REGION Network 7: INITIALIZE ALL STATIONS TIMER
   #tmrInitAllStns(IN := "HMI".settings.kp8.buttons[0].actuate, PT := t#10s);   // TON
   #initAllStns := #tmrInitAllStns.Q;
END_REGION

REGION Network 8: SET DEFAULT TIMERS
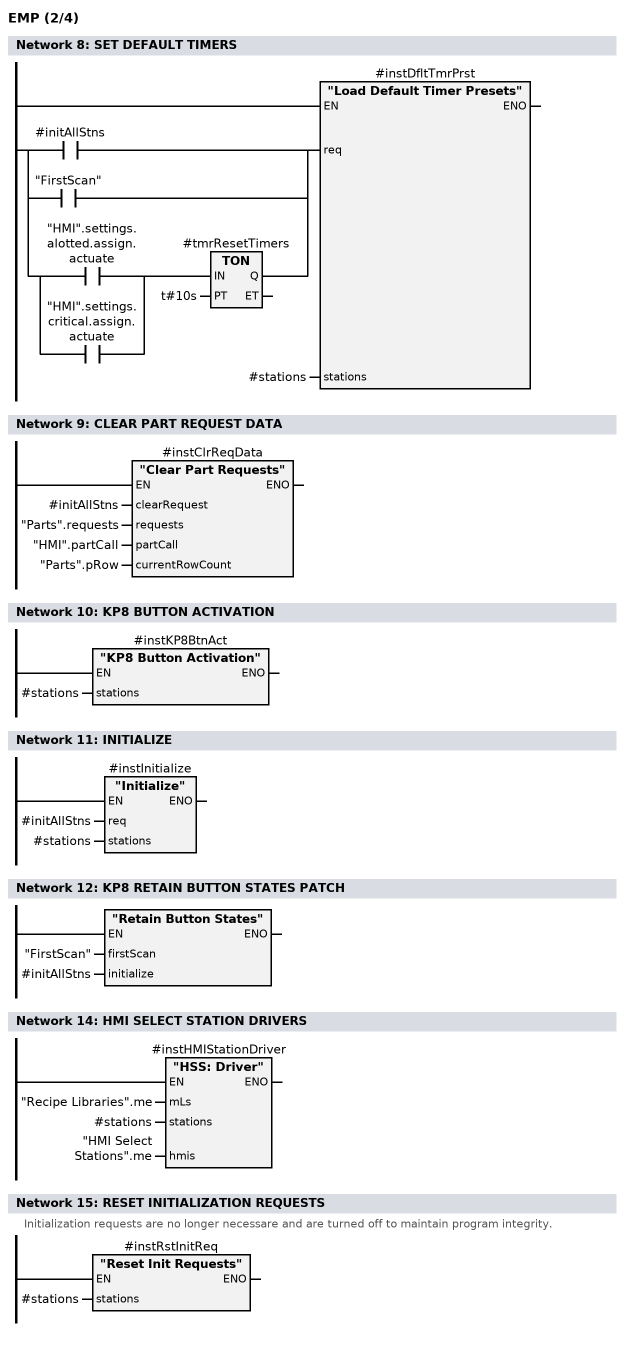
   #tmrResetTimers(IN := "HMI".settings.alotted.assign.actuate OR "HMI".settings.critical.assign.actuate,   // TON
                   PT := t#10s);
   #instDfltTmrPrst(req := #initAllStns OR "FirstScan" OR #tmrResetTimers.Q, stations := #stations);   // "Load Default Timer Presets"
END_REGION

REGION Network 9: CLEAR PART REQUEST DATA
   RUNG wire#powerrail
      #instClrReqData(clearRequest := #initAllStns, requests := "Parts".requests, partCall := "HMI".partCall, currentRowCount := "Parts".pRow)
   END_RUNG
   // the same network as SCL:
   #instClrReqData(clearRequest := #initAllStns,   // "Clear Part Requests"
                   requests := "Parts".requests,
                   partCall := "HMI".partCall,
                   currentRowCount := "Parts".pRow);
END_REGION

REGION Network 10: KP8 BUTTON ACTIVATION
   RUNG wire#powerrail
      #instKP8BtnAct(stations := #stations)
   END_RUNG
   // the same network as SCL:
   #instKP8BtnAct(stations := #stations);   // "KP8 Button Activation"
END_REGION

REGION Network 11: INITIALIZE
   RUNG wire#powerrail
      #instInitialize(req := #initAllStns, stations := #stations)
   END_RUNG
   // the same network as SCL:
   #instInitialize(req := #initAllStns, stations := #stations);   // "Initialize"
END_REGION

REGION Network 12: KP8 RETAIN BUTTON STATES PATCH
   RUNG wire#powerrail
      "Retain Button States"(firstScan := "FirstScan", initialize := #initAllStns)
   END_RUNG
   // the same network as SCL:
   "Retain Button States"(firstScan := "FirstScan", initialize := #initAllStns);
END_REGION

REGION Network 13 (SCL): KP8 DRIVER CALLS
   REGION "LOOP THROUGH STATIONS"
       FOR #i := 0 TO "stnCount" DO
           CASE #i OF
               0..24, 30..38:
                   #instKP8Drvs[#i](btnIn := #stations.me[#i].kp8In,
                                    hardInit := #stations.me[#i].init.hard,
                                    softInit := #stations.me[#i].init.soft,
                                    btn0Activate := #stations.me[#i].kp8Config.activate[0],
                                    btn0Mode := #stations.me[#i].kp8Config.mode[0],
                                    btn0Group := #stations.me[#i].kp8Config.group[0],
                                    btn0Flash := #stations.me[#i].kp8Config.flash[0],
                                    btn0ColorOn1 := #stations.me[#i].kp8Config.colorOn1[0],
                                    btn0ColorOn2 := #stations.me[#i].kp8Config.colorOn2[0],
                                    btn0ColorOff := #stations.me[#i].kp8Config.colorOff[0],
                                    btn1Activate := #stations.me[#i].kp8Config.activate[1],
                                    btn1Mode := #stations.me[#i].kp8Config.mode[1],
                                    btn1Group := #stations.me[#i].kp8Config.group[1],
                                    btn1Flash := #stations.me[#i].kp8Config.flash[1],
                                    btn1ColorOn1 := #stations.me[#i].kp8Config.colorOn1[1],
                                    btn1ColorOn2 := #stations.me[#i].kp8Config.colorOn2[1],
                                    btn1ColorOff := #stations.me[#i].kp8Config.colorOff[1],
                                    btn2Activate := #stations.me[#i].kp8Config.activate[2],
                                    btn2Mode := #stations.me[#i].kp8Config.mode[2],
                                    btn2Group := #stations.me[#i].kp8Config.group[2],
                                    btn2Flash := #stations.me[#i].kp8Config.flash[2],
                                    btn2ColorOn1 := #stations.me[#i].kp8Config.colorOn1[2],
                                    btn2ColorOn2 := #stations.me[#i].kp8Config.colorOn2[2],
                                    btn2ColorOff := #stations.me[#i].kp8Config.colorOff[2],
                                    btn3Activate := #stations.me[#i].kp8Config.activate[3],
                                    btn3Mode := #stations.me[#i].kp8Config.mode[3],
                                    btn3Group := #stations.me[#i].kp8Config.group[3],
                                    btn3Flash := #stations.me[#i].kp8Config.flash[3],
                                    btn3ColorOn1 := #stations.me[#i].kp8Config.colorOn1[3],
                                    btn3ColorOn2 := #stations.me[#i].kp8Config.colorOn2[3],
                                    btn3ColorOff := #stations.me[#i].kp8Config.colorOff[3],
                                    btn4Activate := #stations.me[#i].kp8Config.activate[4],
                                    btn4Mode := #stations.me[#i].kp8Config.mode[4],
                                    btn4Group := #stations.me[#i].kp8Config.group[4],
                                    btn4Flash := #stations.me[#i].kp8Config.flash[4],
                                    btn4ColorOn1 := #stations.me[#i].kp8Config.colorOn1[4],
                                    btn4ColorOn2 := #stations.me[#i].kp8Config.colorOn2[4],
                                    btn4ColorOff := #stations.me[#i].kp8Config.colorOff[4],
                                    btn5Activate := #stations.me[#i].kp8Config.activate[5],
                                    btn5Mode := #stations.me[#i].kp8Config.mode[5],
                                    btn5Group := #stations.me[#i].kp8Config.group[5],
                                    btn5Flash := #stations.me[#i].kp8Config.flash[5],
                                    btn5ColorOn1 := #stations.me[#i].kp8Config.colorOn1[5],
                                    btn5ColorOn2 := #stations.me[#i].kp8Config.colorOn2[5],
                                    btn5ColorOff := #stations.me[#i].kp8Config.colorOff[5],
                                    btn6Activate := #stations.me[#i].kp8Config.activate[6],
                                    btn6Mode := #stations.me[#i].kp8Config.mode[6],
                                    btn6Group := #stations.me[#i].kp8Config.group[6],
                                    btn6Flash := #stations.me[#i].kp8Config.flash[6],
                                    btn6ColorOn1 := #stations.me[#i].kp8Config.colorOn1[6],
                                    btn6ColorOn2 := #stations.me[#i].kp8Config.colorOn2[6],
                                    btn6ColorOff := #stations.me[#i].kp8Config.colorOff[6],
                                    btn7Activate := #stations.me[#i].kp8Config.activate[7],
                                    btn7Mode := #stations.me[#i].kp8Config.mode[7],
                                    btn7Group := #stations.me[#i].kp8Config.group[7],
                                    btn7Flash := #stations.me[#i].kp8Config.flash[7],
                                    btn7ColorOn1 := #stations.me[#i].kp8Config.colorOn1[7],
                                    btn7ColorOn2 := #stations.me[#i].kp8Config.colorOn2[7],
                                    btn7ColorOff := #stations.me[#i].kp8Config.colorOff[7],
                                    btnStatesOut => #stations.me[#i].btnStates,
                                    btnColorsOut => #stations.me[#i].kp8Out);
               ELSE 
                   ;
           END_CASE;

       END_FOR;
   END_REGION
END_REGION

REGION Network 14: HMI SELECT STATION DRIVERS
   RUNG wire#powerrail
      #instHMIStationDriver(mLs := "Recipe Libraries".me, stations := #stations, hmis := "HMI Select Stations".me)
   END_RUNG
   // the same network as SCL:
   #instHMIStationDriver(mLs := "Recipe Libraries".me, stations := #stations, hmis := "HMI Select Stations".me);   // "HSS: Driver"
END_REGION

REGION Network 15: RESET INITIALIZATION REQUESTS
   // Initialization requests are no longer necessare and are turned off to maintain program integrity.
   RUNG wire#powerrail
      #instRstInitReq(stations := #stations)
   END_RUNG
   // the same network as SCL:
   #instRstInitReq(stations := #stations);   // "Reset Init Requests"
END_REGION

REGION Network 16: BARCODE SCREEN
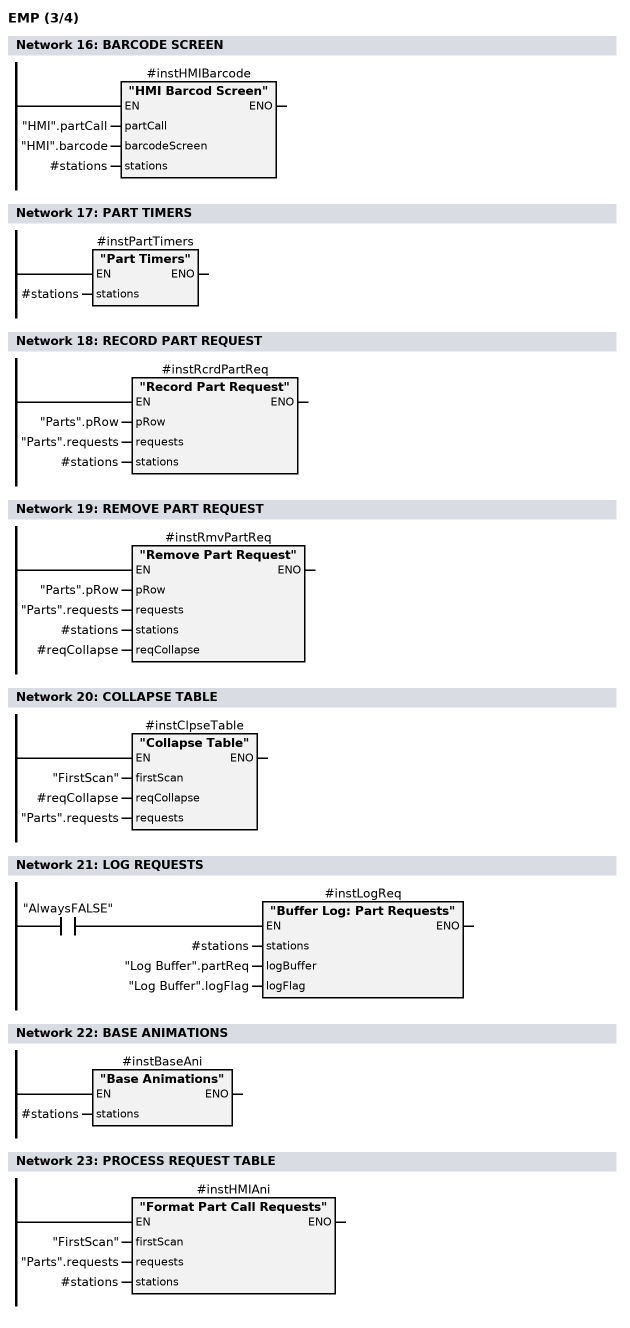
   RUNG wire#powerrail
      #instHMIBarcode(partCall := "HMI".partCall, barcodeScreen := "HMI".barcode, stations := #stations)
   END_RUNG
   // the same network as SCL:
   #instHMIBarcode(partCall := "HMI".partCall, barcodeScreen := "HMI".barcode, stations := #stations);   // "HMI Barcod Screen"
END_REGION

REGION Network 17: PART TIMERS
   RUNG wire#powerrail
      #instPartTimers(stations := #stations)
   END_RUNG
   // the same network as SCL:
   #instPartTimers(stations := #stations);   // "Part Timers"
END_REGION

REGION Network 18: RECORD PART REQUEST
   RUNG wire#powerrail
      #instRcrdPartReq(pRow := "Parts".pRow, requests := "Parts".requests, stations := #stations)
   END_RUNG
   // the same network as SCL:
   #instRcrdPartReq(pRow := "Parts".pRow, requests := "Parts".requests, stations := #stations);   // "Record Part Request"
END_REGION

REGION Network 19: REMOVE PART REQUEST
   RUNG wire#powerrail
      #instRmvPartReq(pRow := "Parts".pRow, requests := "Parts".requests, stations := #stations, reqCollapse := #reqCollapse)
   END_RUNG
   // the same network as SCL:
   #instRmvPartReq(pRow := "Parts".pRow,   // "Remove Part Request"
                   requests := "Parts".requests,
                   stations := #stations,
                   reqCollapse := #reqCollapse);
END_REGION

REGION Network 20: COLLAPSE TABLE
   RUNG wire#powerrail
      #instClpseTable(firstScan := "FirstScan", reqCollapse := #reqCollapse, requests := "Parts".requests)
   END_RUNG
   // the same network as SCL:
   #instClpseTable(firstScan := "FirstScan", reqCollapse := #reqCollapse, requests := "Parts".requests);   // "Collapse Table"
END_REGION

REGION Network 21: LOG REQUESTS
   RUNG wire#powerrail
      Contact( "AlwaysFALSE" )
      #instLogReq(stations := #stations, logBuffer := "Log Buffer".partReq, logFlag := "Log Buffer".logFlag)
   END_RUNG
   // the same network as SCL:
   IF "AlwaysFALSE" THEN
       #instLogReq(stations := #stations, logBuffer := "Log Buffer".partReq, logFlag := "Log Buffer".logFlag);   // "Buffer Log: Part Requests"
   END_IF;
END_REGION

REGION Network 22: BASE ANIMATIONS
   RUNG wire#powerrail
      #instBaseAni(stations := #stations)
   END_RUNG
   // the same network as SCL:
   #instBaseAni(stations := #stations);   // "Base Animations"
END_REGION

REGION Network 23: PROCESS REQUEST TABLE
   RUNG wire#powerrail
      #instHMIAni(firstScan := "FirstScan", requests := "Parts".requests, stations := #stations)
   END_RUNG
   // the same network as SCL:
   #instHMIAni(firstScan := "FirstScan", requests := "Parts".requests, stations := #stations);   // "Format Part Call Requests"
END_REGION

REGION Network 24: HMI POPULATE TABLE
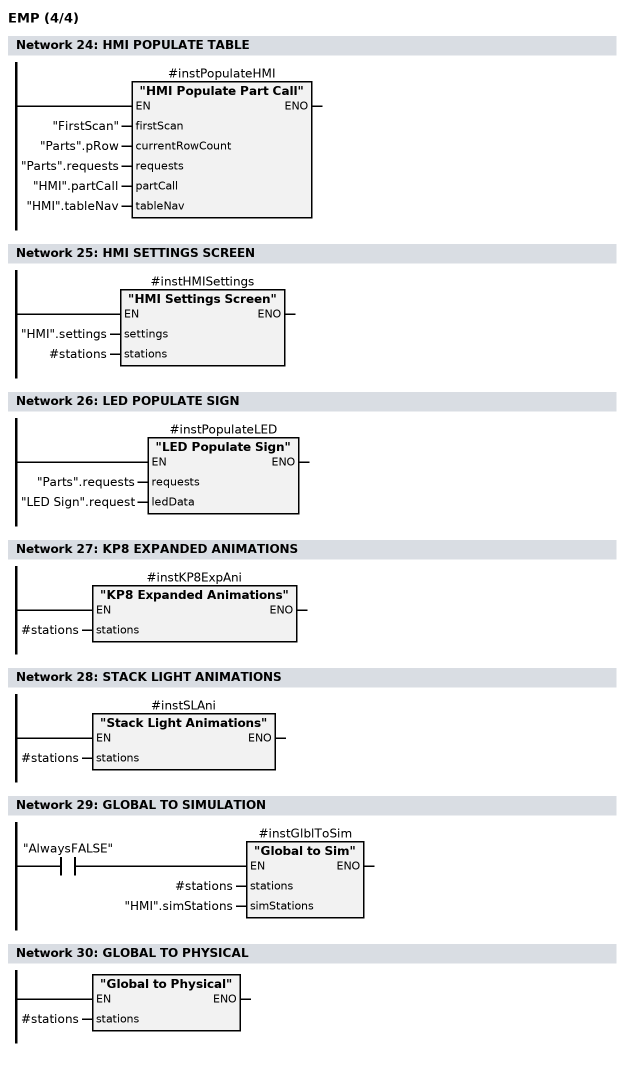
   RUNG wire#powerrail
      #instPopulateHMI(firstScan := "FirstScan", currentRowCount := "Parts".pRow, requests := "Parts".requests, partCall := "HMI".partCall, tableNav := "HMI".tableNav)
   END_RUNG
   // the same network as SCL:
   #instPopulateHMI(firstScan := "FirstScan",   // "HMI Populate Part Call"
                    currentRowCount := "Parts".pRow,
                    requests := "Parts".requests,
                    partCall := "HMI".partCall,
                    tableNav := "HMI".tableNav);
END_REGION

REGION Network 25: HMI SETTINGS SCREEN
   RUNG wire#powerrail
      #instHMISettings(settings := "HMI".settings, stations := #stations)
   END_RUNG
   // the same network as SCL:
   #instHMISettings(settings := "HMI".settings, stations := #stations);   // "HMI Settings Screen"
END_REGION

REGION Network 26: LED POPULATE SIGN
   RUNG wire#powerrail
      #instPopulateLED(requests := "Parts".requests, ledData := "LED Sign".request)
   END_RUNG
   // the same network as SCL:
   #instPopulateLED(requests := "Parts".requests, ledData := "LED Sign".request);   // "LED Populate Sign"
END_REGION

REGION Network 27: KP8 EXPANDED ANIMATIONS
   RUNG wire#powerrail
      #instKP8ExpAni(stations := #stations)
   END_RUNG
   // the same network as SCL:
   #instKP8ExpAni(stations := #stations);   // "KP8 Expanded Animations"
END_REGION

REGION Network 28: STACK LIGHT ANIMATIONS
   RUNG wire#powerrail
      #instSLAni(stations := #stations)
   END_RUNG
   // the same network as SCL:
   #instSLAni(stations := #stations);   // "Stack Light Animations"
END_REGION

REGION Network 29: GLOBAL TO SIMULATION
   RUNG wire#powerrail
      Contact( "AlwaysFALSE" )
      #instGlblToSim(stations := #stations, simStations := "HMI".simStations)
   END_RUNG
   // the same network as SCL:
   IF "AlwaysFALSE" THEN
       #instGlblToSim(stations := #stations, simStations := "HMI".simStations);   // "Global to Sim"
   END_IF;
END_REGION

REGION Network 30: GLOBAL TO PHYSICAL
   RUNG wire#powerrail
      "Global to Physical"(stations := #stations)
   END_RUNG
   // the same network as SCL:
   "Global to Physical"(stations := #stations);
END_REGION
END_FUNCTION_BLOCK

FUNCTION_BLOCK "Code 128"   // FB2, SCL
{ S7_Optimized_Access := 'TRUE' }
VERSION : 0.1
   VAR_INPUT
      partNumber : String;
   END_VAR
   VAR_OUTPUT
      barcode : String;
   END_VAR
   VAR
      charsIn : Array[0..255] of Byte;
      charsOut : Array[0..255] of Byte;
      cnt : UInt;
      intVals : Array[0..255] of Int;
      sum : Int;
      checkSum : Int;
   END_VAR
   VAR_TEMP
      pn : String;
      i : Int;
   END_VAR
   VAR CONSTANT
      startChar : Char := 'Ì';
      stopChar : Char := 'Î';
   END_VAR
   // intVals[0] := 104;
BEGIN
   #pn := #partNumber;

   FOR #i := 0 TO 255 DO
       #charsIn[#i] := 16#00;
       #charsOut[#i] := 16#00;
       #intVals[#i] := 0;
   END_FOR;

   Strg_TO_Chars(Strg:=#pn,
                 pChars:=0,
                 Cnt=>#cnt,
                 Chars:=#charsIn);


   #sum := 104;
   FOR #i := 0 TO UINT_TO_INT(#cnt - 1) DO
       #intVals[#i] := CHAR_TO_INT(#charsIn[#i]) - 32;
       #intVals[#i] := #intVals[#i] * (#i + 1);
       #sum := #sum + #intVals[#i];
   END_FOR;
   #checkSum := (#sum MOD 103) + 32;
   IF #checkSum >= 127 THEN
       #checkSum := #checkSum + 68;
   END_IF;

   #charsOut[0] := #startChar;
   FOR #i := 1 TO UINT_TO_INT(#cnt) DO
       #charsOut[#i] := #charsIn[#i - 1];
   END_FOR;
   #charsOut[#cnt + 1] := INT_TO_BYTE(#checkSum);
   #charsOut[#cnt + 2] := INT_TO_BYTE(#stopChar);

   Chars_TO_Strg(Chars := #charsOut,
                 pChars := 0,
                 Cnt := #cnt + 3,
                 Strg => #barcode);
END_FUNCTION_BLOCK

FUNCTION_BLOCK "HMI Barcod Screen"   // FB3, SCL
{ S7_Optimized_Access := 'TRUE' }
VERSION : 0.1
   VAR_IN_OUT
      partCall : "Part Call Screen";
      barcodeScreen : "Barcode Screen";
      stations : "Stations";
   END_VAR
   VAR
      address : UInt;
      button : UInt;
      instCode128 : "Code 128";
      codeOut : String;
      pnOut : WString[40];
      station : UInt;
      oldSelectedRow : Int;
      oldOrderedBtn : Bool;
   END_VAR
   VAR_TEMP
      orderCancelled : Int;
      processedPN : String[40];
      selectedPN : String[40];
      userOrdered : Bool;
      selectedRow : Int;
      position : Int;
   END_VAR
   VAR CONSTANT
      maxRows : Int := 199;
   END_VAR
BEGIN
   REGION "GET USER ROW SELECTION"
       #selectedRow := "Get Part Call Row Number"(partCall := #partCall); 
   END_REGION

   REGION "ON SELECTION OF A PART CALL ROW
       IF #selectedRow <> 0 THEN
           IF #selectedRow <> #oldSelectedRow THEN

               REGION "GET BUTTON AND STATION NUMBERS"
                   #address := #partCall.row[#selectedRow - 1].address;
                   "Address to Station and Button"(address := #address,
                                                   station => #station,
                                                   button => #button);
               END_REGION

               REGION "CONVERT STRING TO BARCODE"

                   REGION "COPY TO LOCALS"
                       #selectedPN := WSTRING_TO_STRING(#partCall.row[#selectedRow - 1].tfPartNumber.value);
                   END_REGION

                   REGION "CHECK FOR MULTI LINE"

                       REGION "GET POSITON OF CARRIAGE RETURN"
                           #position := FIND(IN1 := #selectedPN, IN2 := '$L');
                       END_REGION

                       REGION "MULTILINE"
                           IF #position <> 0 THEN
                               #processedPN := LEFT(IN := #selectedPN, L := #position - 1);
                           END_IF;
                       END_REGION

                       REGION "SINGLE LINE"
                           IF #position = 0 THEN
                               #processedPN := #selectedPN;
                           END_IF;
                       END_REGION

                   END_REGION

                   REGION "CONVERT TO BARCODE"
                       #instCode128(partNumber := #processedPN,
                                    barcode => #codeOut);
                   END_REGION

                   REGION "OUTPUT FOR HMI SCREEN"
                       #barcodeScreen.partNumber := STRING_TO_WSTRING(#processedPN);
                       #barcodeScreen.barcode := #codeOut;
                   END_REGION

               END_REGION

           END_IF;
       END_IF;
   END_REGION

   REGION "PASS USER ORDERED"

       REGION "COPY TO LOCAL"
           #userOrdered := #barcodeScreen.ordered;
       END_REGION

       REGION "TURN OFF THE LIGHTS"
           #barcodeScreen.ordered := FALSE;
       END_REGION

       REGION "ON RISING EDGE"
           IF #userOrdered AND NOT #oldOrderedBtn THEN

               REGION "SET PART ORDERED"
                   #stations.me[#station - 1].partOrdered[#button - 1] := #userOrdered;
               END_REGION

           END_IF;
       END_REGION

       REGION "CHANGE DETECTION"
           #oldOrderedBtn := #userOrdered;
       END_REGION

   END_REGION

   REGION "CHANGE DETECTION"    
       #oldSelectedRow := #selectedRow;
   END_REGION
END_FUNCTION_BLOCK

FUNCTION_BLOCK "Initialize"   // FB4, SCL
{ S7_Optimized_Access := 'TRUE' }
VERSION : 0.1
   VAR_INPUT
      req : Bool;
   END_VAR
   VAR_IN_OUT
      stations : "Stations";
   END_VAR
   VAR
      rtElapsed : Real;
      rt : "Runtime Data";
   END_VAR
   VAR_TEMP
      i : Int;
      reset : Struct
         req : Bool;
         elapsed : Real;
      END_STRUCT;
      init : Bool;
   END_VAR
   VAR CONSTANT
      resetLimit : Real := 1.25;
   END_VAR
BEGIN
   REGION "FIRST SCAN OR REQUEST"
       IF #req THEN
           // initialize all stations on plc first scan
           FOR #i := 0 TO "stnCount" DO
               #stations.me[#i].init.hard := TRUE;
           END_FOR;
       END_IF;
   END_REGION

   REGION "RUNTIME CALL"
       // get elapsed time
       #rt.elapsed := RUNTIME(#rt.mem);
       // convert to real data type
       #rtElapsed := LREAL_TO_REAL(#rt.elapsed);
   END_REGION

   REGION "BUTTON 0 BASED RESET TIMERS"
       FOR #i := 0 TO "stnCount" DO

           REGION "PRE-CONDITION"
               // init off by default
               #init := FALSE;
               // request is button 0 on kp8
               #reset.req := #stations.me[#i].kp8In.%X0;
               // saved to shorter name
               #reset.elapsed := #stations.me[#i].elapsedTime.resetReq;
           END_REGION

           REGION "RESET REQUEST"
               IF NOT #reset.req THEN
                   #reset.elapsed := 0.0;
               END_IF;
               IF #reset.req THEN
                   // incriment elapsed time
                   #reset.elapsed := #reset.elapsed + #rtElapsed;
                   // timer expired condition
                   IF #reset.elapsed >= #resetLimit THEN
                       #init := TRUE;
                       #reset.elapsed := 0.0;
                   END_IF;
               END_IF;
               // save elapsed time
               #stations.me[#i].elapsedTime.resetReq := #reset.elapsed;
           END_REGION

           REGION "SAVE INITIALIZATIN REQUEST"
               #stations.me[#i].init.hard := #init;
           END_REGION

       END_FOR;
   END_REGION
END_FUNCTION_BLOCK

FUNCTION_BLOCK "Reset Init Requests"   // FB5, SCL
{ S7_Optimized_Access := 'TRUE' }
VERSION : 0.1
   VAR_IN_OUT
      stations : "Stations";
   END_VAR
   VAR
      placeHolder : Bool;
   END_VAR
   VAR_TEMP
      i : Int;
      stnCount : Int;
   END_VAR
BEGIN
   REGION "GET STATION COUNT"
       #stnCount := "stnCount";
   END_REGION

   REGION "RESET INITIALIZATION REQUESTS
       FOR #i := 0 TO #stnCount DO
           #stations.me[#i].init.hard := FALSE;
           #stations.me[#i].init.soft := FALSE;
       END_FOR;
   END_REGION
END_FUNCTION_BLOCK

FUNCTION_BLOCK "Record Part Request"   // FB6, SCL
{ S7_Optimized_Access := 'TRUE' }
VERSION : 0.1
   VAR_IN_OUT
      pRow : Int;
      requests : "Part Request Data";
      stations : "Stations";
   END_VAR
   VAR
      enterAddress : Bool;
      old : Struct
         presses : "Station Old Presses";
      END_STRUCT;
   END_VAR
   VAR_TEMP
      address : UInt;
      hasPart : Bool;
      i : Int;
      j : Int;
      k : Int;
      logAddress : UInt;
      noPart : Bool;
      oldPartReq : Bool;
      partReq : Bool;
      partNumber : WString;
   END_VAR
BEGIN
   REGION "FOR EACH STATION"
       FOR #i := 0 TO "stnCount" DO

           REGION "FOR EACH BUTTON"
               // j = 0 is excluded because it is used as a station reset button
               FOR #j := 1 TO "ptsPerStn" DO

                   REGION "COPY TO LOCAL"
                       #partReq := #stations.me[#i].btnStates[#j];
                       #oldPartReq := #old.presses.me[#i,#j];
                   END_REGION

                   REGION "DETERMINE STATE"

                       REGION "ON NEW REQUEST"
                           IF #partReq AND NOT #oldPartReq THEN

                               REGION "COPY TO LOCAL"
                                   #partNumber := #stations.me[#i].partNumbers[#j];
                               END_REGION

                               REGION "BUTTON HAS NO PN"
                                   IF LEN(#partNumber) = 0 THEN
                                       #hasPart := FALSE;
                                       #noPart := TRUE;
                                   END_IF;
                               END_REGION

                               REGION "BUTTON HAS PN"
                                   IF LEN(#partNumber) <> 0 THEN
                                       #hasPart := TRUE;
                                       #noPart := FALSE;
                                   END_IF;
                               END_REGION

                           END_IF;

                           REGION "SAVE FOR CHANGE DETECTION"
                               #old.presses.me[#i, #j] := #stations.me[#i].btnStates[#j];
                           END_REGION

                       END_REGION

                   END_REGION

                   REGION "NO PART"
                       IF #noPart THEN

                           REGION "TURN OFF THE LIGHTS"
                               #hasPart := FALSE;
                               #noPart := FALSE;
                               #enterAddress := FALSE;
                           END_REGION

                       END_IF;
                   END_REGION

                   REGION "HAS PART"
                       IF #hasPart THEN

                           REGION "TURN OFF THE LIGHTS"
                               #hasPart := FALSE;
                               #noPart := FALSE;
                               #enterAddress := FALSE;
                           END_REGION

                           REGION "CALCULATE ADDRESS"
                               #address := (INT_TO_UINT(#i) + 1) * 10 + (INT_TO_UINT(#j) + 1);
                           END_REGION

                           REGION "SET FLAG"
                               #enterAddress := TRUE;
                           END_REGION

                           REGION "CHECK FOR ENTRY IN DB"
                               REGION "FOR EACH ROW IN PART DB"
                                   FOR #k := 0 TO "partReqDataRowCount" DO

                                       REGION "COPY TO LOCAL"
                                           #logAddress := #requests.row[#k].address;
                                       END_REGION

                                       REGION "RESET FLAG"
                                           IF #logAddress = #address THEN
                                               #enterAddress := FALSE;
                                           END_IF;
                                       END_REGION

                                   END_FOR;
                               END_REGION
                           END_REGION


                       END_IF;
                   END_REGION

                   REGION "SAVE ROW DATA"
                       IF #enterAddress THEN

                           REGION "TURN OFF THE LIGHTS"
                               #enterAddress := FALSE;
                           END_REGION

                           REGION "ENTER PART REQUEST"
                               #stations.me[#i].partRequested[#j] := TRUE;
                           END_REGION

                           REGION "ADDRESS"
                               #requests.row[#pRow].address := #address;
                           END_REGION

                           REGION "LINE"
                               #requests.row[#pRow].tfLine.value := #stations.me[#i].line;
                           END_REGION

                           REGION "DROP ZONE"
                               #requests.row[#pRow].tfDropZone.value := USINT_TO_WSTRING(#stations.me[#i].dropZone);
                           END_REGION

                           REGION "PART NUMBER"
                               #requests.row[#pRow].tfPartNumber.value := #stations.me[#i].partNumbers[#j];
                           END_REGION

                           REGION "ELLAPSED TIME"
                               #requests.row[#pRow].tfTime.value := "Real to WString Timer"(#stations.me[#i].elapsedTime.partReq[#j]);
                           END_REGION

                           REGION "ROW POINTER"

                               REGION "INCREMENT"
                                   #pRow := #pRow + 1;
                               END_REGION

                               REGION "HIGH LIMIT ROLLOVER"
                                   IF #pRow > "partReqDataRowCount" THEN
                                       #pRow := 0;
                                   END_IF;
                               END_REGION

                           END_REGION

                       END_IF;
                   END_REGION

               END_FOR;
           END_REGION

       END_FOR;
   END_REGION
END_FUNCTION_BLOCK

FUNCTION_BLOCK "Part Timers"   // FB7, SCL
{ S7_Optimized_Access := 'TRUE' }
VERSION : 0.1
   VAR_IN_OUT
      stations : "Stations";
   END_VAR
   VAR
      rt : "Runtime Data";
      old : Struct
         presses : "Station Old Presses";
      END_STRUCT;
   END_VAR
   VAR_TEMP
      alottedTime : Real;
      btnCount : Int;
      elapsedTime : Real;
      i : Int;
      j : Int;
      partRequested : Bool;
      redTime : Real;
      remainingTime : Real;
      stnCount : Int;
      press : Struct
         current : Bool;
         old : Bool;
      END_STRUCT;
   END_VAR
BEGIN
   REGION "RUNTIME CALL"
       #rt.elapsed := RUNTIME(#rt.mem);
       #rt.asReal := LREAL_TO_REAL(#rt.elapsed);
   END_REGION

   REGION "COPY TO LOCAL"
       #stnCount := "stnCount";
       #btnCount := "ptsPerStn";
   END_REGION

   REGION "FOR EACH STATION"
       FOR #i := 0 TO #stnCount DO

           REGION "FOR EACH BUTTON"
               // j := 0 would be the reset button so it is skipped
               FOR #j := 1 TO #btnCount DO

                   REGION "RESET PART TIMER"

                       REGION "COPY TO LOCAL"
                           #press.current := #stations.me[#i].btnStates[#j];
                           #press.old := #old.presses.me[#i, #j];
                       END_REGION

                       REGION "ON PRESS FALLING EDGE"
                           IF NOT #press.current AND #press.old THEN
                               #stations.me[#i].elapsedTime.partReq[#j] := 0.0;
                           END_IF;
                           #old.presses.me[#i, #j] := #stations.me[#i].btnStates[#j];
                       END_REGION

                   END_REGION

                   REGION "PART REQUEST TIMER"

                       REGION "COPY TO LOCAL"
                           #partRequested := #stations.me[#i].btnStates[#j];
                       END_REGION

                       REGION "ON PART REQUEST"
                           IF #partRequested THEN

                               REGION "OUTPUT ELLAPSED TIME"
                                   // get saved time
                                   #elapsedTime := #stations.me[#i].elapsedTime.partReq[#j];
                                   // add elapsed time
                                   #elapsedTime += #rt.asReal;
                                   // save new value
                                   #stations.me[#i].elapsedTime.partReq[#j] := #elapsedTime;
                               END_REGION

                           END_IF;
                       END_REGION

                   END_REGION

               END_FOR;
           END_REGION

       END_FOR;
   END_REGION
END_FUNCTION_BLOCK

FUNCTION_BLOCK "Base Animations"   // FB8, SCL
{ S7_Optimized_Access := 'TRUE' }
VERSION : 0.1
   VAR_IN_OUT
      stations : "Stations";
   END_VAR
   VAR_TEMP
      animation : Int;
      i : Int;
      j : Int;
      partRequested : Bool;
      partOrdered : Bool;
      elapsedTime : Real;
      criticalTime : Real;
      alottedTime : Real;
      remainingTime : Real;
      stnCount : Int;
   END_VAR
   VAR CONSTANT
      anDefault : USInt := 0;
      anRequested : USInt := 1;
      anSolidRed : USInt := 2;
      anFlashRed : USInt := 3;
      anPartOrdered : USInt := 4;
   END_VAR
BEGIN
   REGION "COPY TO LOCAL"
       #stnCount := "stnCount";
   END_REGION

   REGION "FOR EACH STATION"
       FOR #i := 0 TO #stnCount DO

           REGION "FOR EACH BUTTON"
               // j := 0 would be the reset button so it is skipped
               FOR #j := 1 TO 7 DO

                   REGION "PART REQUEST TIMER"

                       REGION "COPY TO LOCAL"
                           #partRequested := #stations.me[#i].btnStates[#j];
                           #partOrdered := #stations.me[#i].partOrdered[#j];
                       END_REGION

                       REGION "PART REQUESTED"
                           IF #partRequested THEN

                               REGION "COPY TO LOCAL"
                                   // remaining time
                                   #elapsedTime := #stations.me[#i].elapsedTime.partReq[#j];
                                   #alottedTime := #stations.me[#i].presetTime.allotted[#j];
                                   #remainingTime := #alottedTime - #elapsedTime;
                                   // critical time
                                   #criticalTime := #stations.me[#i].presetTime.critical[#j];
                               END_REGION

                               REGION "DEFAULT ANIMATION STATE"
                                   IF #remainingTime > #criticalTime THEN
                                       #animation := #anRequested;
                                   END_IF;
                               END_REGION

                               REGION "ORDERED"
                                   IF #partOrdered THEN
                                       #animation := #anPartOrdered;
                                   END_IF;
                               END_REGION

                               REGION "SOLID RED ANIMATION STATE"
                                   IF #remainingTime <= #criticalTime AND #elapsedTime > 0.0 THEN
                                       #animation := #anSolidRed;
                                   END_IF;
                               END_REGION

                               REGION "FLASHING RED ANIMATION STATE
                                   IF #remainingTime <= 0.0 THEN
                                       #animation := #anFlashRed;
                                   END_IF;
                               END_REGION

                           END_IF;
                       END_REGION

                       REGION "PART NOT REQUESTED"
                           IF NOT #partRequested THEN
                               #animation := #anDefault;
                           END_IF;
                       END_REGION

                       REGION "OUTPUT"
                           #stations.me[#i].animations[#j] := #animation;
                       END_REGION

                   END_REGION

               END_FOR;
           END_REGION

       END_FOR;
   END_REGION
END_FUNCTION_BLOCK

FUNCTION_BLOCK "Format Part Call Requests"   // FB9, SCL
{ S7_Optimized_Access := 'TRUE' }
VERSION : 0.1
   VAR_INPUT
      firstScan : Bool;
   END_VAR
   VAR_IN_OUT
      requests : "Part Request Data";
      stations : "Stations";
   END_VAR
   VAR
      station : Int;
      button : Int;
   END_VAR
   VAR_TEMP
      address : Int;
      animate : USInt;
      timeAsReal : Real;
      timeAsTime : WString;
      i : Int;
      inStrRslt : Int;
      invisible : USInt;
      genericVisible : USInt;
      gray : USInt;
      darkGray : USInt;
      red : USInt;
      blue : USInt;
      redFlashing : USInt;
   END_VAR
   VAR CONSTANT
      visible : USInt := 1;
      anDefault : USInt := 0;
      anRequested : USInt := 1;
      anSolidRed : USInt := 2;
      anFlashRed : USInt := 3;
      anPartOrdered : USInt := 4;
   END_VAR
BEGIN
   REGION "COPY TO LOCAL"
       #invisible := "invisible";
       #gray := "BgGray";
       #darkGray := "disabled";
       #blue := "BgLBl";
       #red := "BgDRd";
       #redFlashing := "FlDrd";
   END_REGION


   REGION "ITERATE THROUGH VISIBLE TABLE ROWS"
       FOR #i := 0 TO "partReqDataRowCount" DO

           REGION "COPY TO LOCAL"
               #address := UINT_TO_INT(#requests.row[#i].address);
           END_REGION

           REGION "HIDE UNPOPULATED ROWS"
               IF #address = 0 THEN
                   #requests.row[#i].pbSelection.animate := #invisible;
                   #requests.row[#i].rtBackground.animate := #invisible;
                   #animate := 0;
                   #requests.row[#i].tfDropZone.animate := #invisible;
                   #requests.row[#i].tfLine.animate := #invisible;
                   #requests.row[#i].tfPartNumber.animateSL := #invisible;
                   #requests.row[#i].tfPartNumber.animateDL := #invisible;
                   #requests.row[#i].tfTime.animate := #invisible;
               END_IF;
           END_REGION

           REGION "ANIMATE POPULATED ROWS"

               REGION "ANIMATE ROWS WITH DATA"
                   IF #address <> 0 THEN

                       REGION "GET POINTERS FOR STATION ARRAY"
                           #station := #address / 10 - 1;
                           #button := #address MOD 10 - 1;
                       END_REGION

                       REGION "SET ANIMATE"
                           CASE #stations.me[#station].animations[#button] OF
                               #anRequested:
                                   #animate := #gray;
                               #anSolidRed:
                                   #animate := #red;
                               #anFlashRed:
                                   #animate := #redFlashing;
                               #anPartOrdered:
                                   #animate := #blue;
                               ELSE
                                   #animate := #invisible;
                           END_CASE;
                       END_REGION


                       REGION "ANIMATIONS"

                           REGION "PUSHBUTTON VISIBILITY"
                               #requests.row[#i].pbSelection.animate := #visible;
                           END_REGION

                           REGION "BACKGROUND VISIBILITY"
                               #requests.row[#i].rtBackground.animate := #darkGray;
                           END_REGION

                           REGION "DROP ZONE" 
                               #requests.row[#i].tfDropZone.animate := #animate;
                               #requests.row[#i].tfDropZone.value := "Strip Sign"(UINT_TO_WSTRING(#stations.me[#station].dropZone));
                           END_REGION

                           REGION "LINE"
                               #requests.row[#i].tfLine.animate := #animate;
                               #requests.row[#i].tfLine.value := #stations.me[#station].line;
                           END_REGION

                           REGION "PART NUMBER"
                               #requests.row[#i].tfPartNumber.animateSL := #animate;
                               #requests.row[#i].tfPartNumber.value := #stations.me[#station].partNumbers[#button];
                               REGION "DETERMINE VISIBLE ROWS"

                                   REGION "FIND CARRIAGE RETURN"
                                       #inStrRslt := FIND(IN1 := #requests.row[#i].tfPartNumber.value,
                                                          IN2 := wstring#'$L');
                                   END_REGION

                                   REGION "SINGLE LINE"
                                       IF #inStrRslt = 0 THEN
                                           #requests.row[#i].tfPartNumber.animateSL := #animate;
                                           #requests.row[#i].tfPartNumber.animateDL := #invisible;
                                       END_IF;
                                   END_REGION

                                   REGION "DOUBLE LINE"
                                       IF #inStrRslt <> 0 THEN
                                           #requests.row[#i].tfPartNumber.animateSL := #invisible;
                                           #requests.row[#i].tfPartNumber.animateDL := #animate;
                                       END_IF;
                                   END_REGION

                               END_REGION

                           END_REGION

                           REGION "TIME"
                               #requests.row[#i].tfTime.animate := #animate;
                               #timeAsReal := #stations.me[#station].presetTime.allotted[#button];
                               #timeAsReal -= #stations.me[#station].elapsedTime.partReq[#button];
                               #requests.row[#i].tfTime.value := "Real to WString Timer"(#timeAsReal);
                           END_REGION

                       END_REGION

                   END_IF;
               END_REGION

           END_REGION

       END_FOR;
   END_REGION
END_FUNCTION_BLOCK

FUNCTION_BLOCK "KP8 Expanded Animations"   // FB10, SCL
{ S7_Optimized_Access := 'TRUE' }
VERSION : 0.1
   VAR_IN_OUT
      stations : "Stations";
   END_VAR
   VAR_TEMP
      i : Int;
      j : Int;
      colorBox : DWord;
      animation : Int;
      mask : DWord;
   END_VAR
   VAR CONSTANT
      anSolidRed : USInt := 2;
      anFlashRed : USInt := 3;
      anBlue : USInt := 4;
   END_VAR
BEGIN
   REGION "LOOP THROUGH STATIONS"
       FOR #i := 0 TO "stnCount" DO

           REGION "LOOP THROUGH BUTTONS"
               FOR #j := 0 TO "ptsPerStn" DO

                   REGION "GET ANIMATION"
                       #animation := #stations.me[#i].animations[#j];
                   END_REGION

                   REGION "SOLID RED"
                       IF #animation = #anSolidRed THEN
                           #colorBox := #stations.me[#i].kp8Out;
                           #mask := 16#FEFEFEFF;
                           #mask := ROL_DWORD(IN := #mask,
                                                 N := INT_TO_UINT(#j));
                           #colorBox := #colorBox AND #mask;
                           #mask := 16#100_0000;
                           #mask := ROL_DWORD(IN := #mask,
                                                 N := INT_TO_UINT(#j));
                           #colorBox := #colorBox OR #mask;
                           #stations.me[#i].kp8Out := #colorBox;
                       END_IF;
                   END_REGION

                   REGION "FLASHING RED"
                       IF #animation = #anFlashRed THEN

                           REGION "RED ON"
                               IF "Clock_1Hz" THEN
                                   #colorBox := #stations.me[#i].kp8Out;
                                   #mask := 16#FEFEFEFF;
                                   #mask := ROL_DWORD(IN := #mask,
                                                         N := INT_TO_UINT(#j));
                                   #colorBox := #colorBox AND #mask;
                                   #mask := 16#100_0000;
                                   #mask := ROL_DWORD(IN := #mask,
                                                         N := INT_TO_UINT(#j));
                                   #colorBox := #colorBox OR #mask;
                                   #stations.me[#i].kp8Out := #colorBox;
                               END_IF;
                           END_REGION

                           REGION "RED OFF"
                               IF NOT "Clock_1Hz" THEN
                                   #colorBox := #stations.me[#i].kp8Out;
                                   #mask := 16#FEFEFEFF;
                                   #mask := ROL_DWORD(IN := #mask,
                                                         N := INT_TO_UINT(#j));
                                   #colorBox := #colorBox AND #mask;
                                   #stations.me[#i].kp8Out := #colorBox;
                               END_IF;
                           END_REGION

                       END_IF;
                   END_REGION

                   REGION "BLUE"
                       IF #animation = #anBlue THEN
                           #colorBox := #stations.me[#i].kp8Out;
                           #mask := 16#FEFEFEFF;
                           #mask := ROL_DWORD(IN := #mask,
                                              N := INT_TO_UINT(#j));
                           #colorBox := #colorBox AND #mask;
                           #mask := 16#0000_0100;
                           #mask := ROL_DWORD(IN := #mask,
                                                 N := INT_TO_UINT(#j));
                           #colorBox := #colorBox OR #mask;
                           #stations.me[#i].kp8Out := #colorBox;
                       END_IF;
                   END_REGION

               END_FOR;
           END_REGION

       END_FOR;
   END_REGION
END_FUNCTION_BLOCK

FUNCTION_BLOCK "Stack Light Animations"   // FB11, SCL
{ S7_Optimized_Access := 'TRUE' }
VERSION : 0.1
   VAR_IN_OUT
      stations : "Stations";
   END_VAR
   VAR_TEMP
      animation : Int;
      i : Int;
      j : Int;
      stackLight : DWord;
   END_VAR
   VAR CONSTANT
      anDefault : USInt := 0;
      anRequested : USInt := 1;
      anSolidRed : USInt := 2;
      anFlashRed : USInt := 3;
      anPartOrdered : USInt := 4;
      buttonCount : Int := 7;
      "Part 01" : Int := 7;
      "Part 01 Green On" : DWord := 16#0400_0000;
      "Part 01 Red On" : DWord := 16#0100_0000;
      "Part 01 Yellow On" : DWord := 16#0200_0000;
      "Part 02" : Int := 3;
      "Part 02 Green On" : DWord := 16#2000_0000;
      "Part 02 Red On" : DWord := 16#0800_0000;
      "Part 02 Yellow On" : DWord := 16#1000_0000;
      "Part 03" : Int := 6;
      "Part 03 Green On" : DWord := 16#0001_0000;
      "Part 03 Red On" : DWord := 16#4000_0000;
      "Part 03 Yellow On" : DWord := 16#8000_0000;
      "Part 04" : Int := 2;
      "Part 04 Green On" : DWord := 16#0008_0000;
      "Part 04 Yellow On" : DWord := 16#0004_0000;
      "Part 04 Red On" : DWord := 16#0002_0000;
      "Part 05" : Int := 5;
      "Part 05 Green On" : DWord := 16#0040_0000;
      "Part 05 Red On" : DWord := 16#0010_0000;
      "Part 05 Yellow On" : DWord := 16#0020_0000;
      "Part 06" : Int := 1;
      "Part 06 Green On" : DWord := 16#0000_0200;
      "Part 06 Red On" : DWord := 16#0080_0000;
      "Part 06 Yellow On" : DWord := 16#0000_0100;
   END_VAR
BEGIN
   REGION "LOOP THROUGH STATIONS"
       FOR #i := 0 TO "stnCount" DO

           REGION "LOOP THROUGH BUTTONS"
               FOR #j := 0 TO #buttonCount DO

                   REGION "COPY INTO LOCAL"
                       #stackLight := #stations.me[#i].stackLightOut;
                       #animation := #stations.me[#i].animations[#j];
                   END_REGION

                   REGION "GREEN"
                       IF #animation = #anDefault THEN
                           CASE #j OF
                               #"Part 01":
                                   #stackLight := #stackLight AND (NOT #"Part 01 Red On");
                                   #stackLight := #stackLight AND (NOT #"Part 01 Yellow On");
                                   #stackLight := #stackLight OR #"Part 01 Green On";
                               #"Part 02":
                                   #stackLight := #stackLight AND (NOT #"Part 02 Red On");
                                   #stackLight := #stackLight AND (NOT #"Part 02 Yellow On");
                                   #stackLight := #stackLight OR #"Part 02 Green On";
                               #"Part 03":
                                   #stackLight := #stackLight AND (NOT #"Part 03 Red On");
                                   #stackLight := #stackLight AND (NOT #"Part 03 Yellow On");
                                   #stackLight := #stackLight OR #"Part 03 Green On";
                               #"Part 04":
                                   #stackLight := #stackLight AND (NOT #"Part 04 Red On");
                                   #stackLight := #stackLight AND (NOT #"Part 04 Yellow On");
                                   #stackLight := #stackLight OR #"Part 04 Green On";
                               #"Part 05":
                                   #stackLight := #stackLight AND (NOT #"Part 05 Red On");
                                   #stackLight := #stackLight AND (NOT #"Part 05 Yellow On");
                                   #stackLight := #stackLight OR #"Part 05 Green On";
                               #"Part 06":
                                   #stackLight := #stackLight AND (NOT #"Part 06 Red On");
                                   #stackLight := #stackLight AND (NOT #"Part 06 Yellow On");
                                   #stackLight := #stackLight OR #"Part 06 Green On";
                               ELSE
                                   ;
                           END_CASE;
                       END_IF;
                   END_REGION

                   REGION "OFF"
                       IF #stations.me[#i].partNumbers[#j] = WSTRING#'' THEN
                           CASE #j OF
                               #"Part 01":
                                   #stackLight := #stackLight AND (NOT #"Part 01 Red On");
                                   #stackLight := #stackLight AND (NOT #"Part 01 Yellow On");
                                   #stackLight := #stackLight AND (NOT #"Part 01 Green On");
                               #"Part 02":
                                   #stackLight := #stackLight AND (NOT #"Part 02 Red On");
                                   #stackLight := #stackLight AND (NOT #"Part 02 Yellow On");
                                   #stackLight := #stackLight AND (NOT #"Part 02 Green On");
                               #"Part 03":
                                   #stackLight := #stackLight AND (NOT #"Part 03 Red On");
                                   #stackLight := #stackLight AND (NOT #"Part 03 Yellow On");
                                   #stackLight := #stackLight AND (NOT #"Part 03 Green On");
                               #"Part 04":
                                   #stackLight := #stackLight AND (NOT #"Part 04 Red On");
                                   #stackLight := #stackLight AND (NOT #"Part 04 Yellow On");
                                   #stackLight := #stackLight AND (NOT #"Part 04 Green On");
                               #"Part 05":
                                   #stackLight := #stackLight AND (NOT #"Part 05 Red On");
                                   #stackLight := #stackLight AND (NOT #"Part 05 Yellow On");
                                   #stackLight := #stackLight AND (NOT #"Part 05 Green On");
                               #"Part 06":
                                   #stackLight := #stackLight AND (NOT #"Part 06 Red On");
                                   #stackLight := #stackLight AND (NOT #"Part 06 Yellow On");
                                   #stackLight := #stackLight AND (NOT #"Part 06 Green On");
                               ELSE
                                   ;
                           END_CASE;
                       END_IF;
                   END_REGION

                   REGION "YELLOW"
                       IF #animation = #anRequested THEN
                           CASE #j OF
                               #"Part 01":
                                   #stackLight := #stackLight AND (NOT #"Part 01 Red On");
                                   #stackLight := #stackLight OR #"Part 01 Yellow On";
                                   #stackLight := #stackLight AND (NOT #"Part 01 Green On");
                               #"Part 02":
                                   #stackLight := #stackLight AND (NOT #"Part 02 Red On");
                                   #stackLight := #stackLight OR #"Part 02 Yellow On";
                                   #stackLight := #stackLight AND (NOT #"Part 02 Green On");
                               #"Part 03":
                                   #stackLight := #stackLight AND (NOT #"Part 03 Red On");
                                   #stackLight := #stackLight OR #"Part 03 Yellow On";
                                   #stackLight := #stackLight AND (NOT #"Part 03 Green On");
                               #"Part 04":
                                   #stackLight := #stackLight AND (NOT #"Part 04 Red On");
                                   #stackLight := #stackLight OR #"Part 04 Yellow On";
                                   #stackLight := #stackLight AND (NOT #"Part 04 Green On");
                               #"Part 05":
                                   #stackLight := #stackLight AND (NOT #"Part 05 Red On");
                                   #stackLight := #stackLight OR #"Part 05 Yellow On";
                                   #stackLight := #stackLight AND (NOT #"Part 05 Green On");
                               #"Part 06":
                                   #stackLight := #stackLight AND (NOT #"Part 06 Red On");
                                   #stackLight := #stackLight OR #"Part 06 Yellow On";
                                   #stackLight := #stackLight AND (NOT #"Part 06 Green On");
                               ELSE
                                   ;
                           END_CASE;
                       END_IF;
                   END_REGION

                   REGION "SOLID RED"
                       IF #animation = #anSolidRed THEN
                           CASE #j OF
                               #"Part 01":
                                   #stackLight := #stackLight OR #"Part 01 Red On";
                                   #stackLight := #stackLight AND (NOT #"Part 01 Yellow On");
                                   #stackLight := #stackLight AND (NOT #"Part 01 Green On");
                               #"Part 02":
                                   #stackLight := #stackLight OR #"Part 02 Red On";
                                   #stackLight := #stackLight AND (NOT #"Part 02 Yellow On");
                                   #stackLight := #stackLight AND (NOT #"Part 02 Green On");
                               #"Part 03":
                                   #stackLight := #stackLight OR #"Part 03 Red On";
                                   #stackLight := #stackLight AND (NOT #"Part 03 Yellow On");
                                   #stackLight := #stackLight AND (NOT #"Part 03 Green On");
                               #"Part 04":
                                   #stackLight := #stackLight OR #"Part 04 Red On";
                                   #stackLight := #stackLight AND (NOT #"Part 04 Yellow On");
                                   #stackLight := #stackLight AND (NOT #"Part 04 Green On");
                               #"Part 05":
                                   #stackLight := #stackLight OR #"Part 05 Red On";
                                   #stackLight := #stackLight AND (NOT #"Part 05 Yellow On");
                                   #stackLight := #stackLight AND (NOT #"Part 05 Green On");
                               #"Part 06":
                                   #stackLight := #stackLight OR #"Part 06 Red On";
                                   #stackLight := #stackLight AND (NOT #"Part 06 Yellow On");
                                   #stackLight := #stackLight AND (NOT #"Part 06 Green On");
                               ELSE
                                   ;
                           END_CASE;
                       END_IF;
                   END_REGION

                   REGION "FLASHING RED"
                       IF #animation = #anFlashRed THEN

                           REGION "RED ON"
                               IF "Clock_1Hz" THEN
                                   CASE #j OF
                                       #"Part 01":
                                           #stackLight := #stackLight OR #"Part 01 Red On";
                                           #stackLight := #stackLight AND (NOT #"Part 01 Yellow On");
                                           #stackLight := #stackLight AND (NOT #"Part 01 Green On");
                                       #"Part 02":
                                           #stackLight := #stackLight OR #"Part 02 Red On";
                                           #stackLight := #stackLight AND (NOT #"Part 02 Yellow On");
                                           #stackLight := #stackLight AND (NOT #"Part 02 Green On");
                                       #"Part 03":
                                           #stackLight := #stackLight OR #"Part 03 Red On";
                                           #stackLight := #stackLight AND (NOT #"Part 03 Yellow On");
                                           #stackLight := #stackLight AND (NOT #"Part 03 Green On");
                                       #"Part 04":
                                           #stackLight := #stackLight OR #"Part 04 Red On";
                                           #stackLight := #stackLight AND (NOT #"Part 04 Yellow On");
                                           #stackLight := #stackLight AND (NOT #"Part 04 Green On");
                                       #"Part 05":
                                           #stackLight := #stackLight OR #"Part 05 Red On";
                                           #stackLight := #stackLight AND (NOT #"Part 05 Yellow On");
                                           #stackLight := #stackLight AND (NOT #"Part 05 Green On");
                                       #"Part 06":
                                           #stackLight := #stackLight OR #"Part 06 Red On";
                                           #stackLight := #stackLight AND (NOT #"Part 06 Yellow On");
                                           #stackLight := #stackLight AND (NOT #"Part 06 Green On");
                                       ELSE
                                           ;
                                   END_CASE;
                               END_IF;
                           END_REGION

                           REGION "RED OFF"
                               IF NOT "Clock_1Hz" THEN
                                   CASE #j OF
                                       #"Part 01":
                                           #stackLight := #stackLight AND (NOT #"Part 01 Red On");
                                           #stackLight := #stackLight AND (NOT #"Part 01 Yellow On");
                                           #stackLight := #stackLight AND (NOT #"Part 01 Green On");
                                       #"Part 02":
                                           #stackLight := #stackLight AND (NOT #"Part 02 Red On");
                                           #stackLight := #stackLight AND (NOT #"Part 02 Yellow On");
                                           #stackLight := #stackLight AND (NOT #"Part 02 Green On");
                                       #"Part 03":
                                           #stackLight := #stackLight AND (NOT #"Part 03 Red On");
                                           #stackLight := #stackLight AND (NOT #"Part 03 Yellow On");
                                           #stackLight := #stackLight AND (NOT #"Part 03 Green On");
                                       #"Part 04":
                                           #stackLight := #stackLight AND (NOT #"Part 04 Red On");
                                           #stackLight := #stackLight AND (NOT #"Part 04 Yellow On");
                                           #stackLight := #stackLight AND (NOT #"Part 04 Green On");
                                       #"Part 05":
                                           #stackLight := #stackLight AND (NOT #"Part 05 Red On");
                                           #stackLight := #stackLight AND (NOT #"Part 05 Yellow On");
                                           #stackLight := #stackLight AND (NOT #"Part 05 Green On");
                                       #"Part 06":
                                           #stackLight := #stackLight AND (NOT #"Part 06 Red On");
                                           #stackLight := #stackLight AND (NOT #"Part 06 Yellow On");
                                           #stackLight := #stackLight AND (NOT #"Part 06 Green On");
                                       ELSE
                                           ;
                                   END_CASE;
                               END_IF;
                           END_REGION

                       END_IF;
                   END_REGION

                   REGION "COPY OUT TO GLOBAL"
                       #stations.me[#i].stackLightOut := #stackLight;
                   END_REGION

               END_FOR;
           END_REGION

       END_FOR;
   END_REGION
END_FUNCTION_BLOCK

FUNCTION_BLOCK "KP8 Button Activation"   // FB12, SCL
{ S7_Optimized_Access := 'TRUE' }
VERSION : 0.1
   VAR_IN_OUT
      stations : "Stations";
   END_VAR
   VAR
      old : Struct
         kp8Config : Array[0.."stnCount"] of "KP8 Button Config";
      END_STRUCT;
   END_VAR
   VAR_TEMP
      currentPNs : Array[0..7] of WString[40];
      i : Int;
      init : Bool;
      j : Int;
      temp : Int;
   END_VAR
BEGIN
   REGION "LOOP THROUGH STATIONS"
       FOR #i := 0 TO "stnCount" DO

           REGION "COPY TO LOCAL"
               #currentPNs := #stations.me[#i].partNumbers;
           END_REGION


           REGION "LOOP THROUGH BUTTONS"
               FOR #j := 0 TO "ptsPerStn" DO

                       REGION "ACTIVATE BUTTON"
                           IF LEN(#currentPNs[#j]) <> 0 THEN
                               #stations.me[#i].kp8Config.activate[#j] := TRUE;
                               #stations.me[#i].kp8Config.colorOff[#j] := 'green';
                               #stations.me[#i].kp8Config.colorOn1[#j] := 'yellow';
                               #stations.me[#i].kp8Config.colorOn2[#j] := '';
                               #stations.me[#i].kp8Config.flash[#j] := FALSE;
                               #stations.me[#i].kp8Config.group[#j] := 0;
                               #stations.me[#i].kp8Config.mode[#j] := TRUE;
                           END_IF;
                       END_REGION

                       REGION "DEACTIVATE BUTTON"
                           IF LEN(#currentPNs[#j]) = 0 THEN
                               #stations.me[#i].kp8Config.activate[#j] := FALSE;
                               #stations.me[#i].kp8Config.colorOff[#j] := 'off';
                               #stations.me[#i].kp8Config.colorOn1[#j] := 'off';
                               #stations.me[#i].kp8Config.colorOn2[#j] := 'off';
                               #stations.me[#i].kp8Config.flash[#j] := FALSE;
                               #stations.me[#i].kp8Config.group[#j] := 0;
                               #stations.me[#i].kp8Config.mode[#j] := FALSE;
                           END_IF;
                       END_REGION

               END_FOR;
           END_REGION

           REGION "SOFT INIT"
               IF #stations.me[#i].kp8Config <> #old.kp8Config[#i] THEN
                   #stations.me[#i].init.soft := TRUE;
               END_IF;
           END_REGION

           REGION "SAVE FOR CHANGE DETECTION"
               #old.kp8Config[#i] := #stations.me[#i].kp8Config;
           END_REGION

       END_FOR;
   END_REGION
END_FUNCTION_BLOCK

FUNCTION_BLOCK "Remove Part Request"   // FB13, SCL
{ S7_Optimized_Access := 'TRUE' }
VERSION : 0.1
   VAR_IN_OUT
      pRow : Int;
      requests : "Part Request Data";
      stations : "Stations";
      reqCollapse : Bool;
   END_VAR
   VAR
      old : Struct
         partReq : "Station Old Presses";
      END_STRUCT;
   END_VAR
   VAR_TEMP
      address : UInt;
      blankRow : "Table Row";
      hasPart : Bool;
      i : Int;
      j : Int;
      k : Int;
      logAddress : UInt;
      noPart : Bool;
      oldPartReq : Bool;
      partNumber : WString;
      partReq : Bool;
      pRemoveRow : Int;
      removeAddress : Bool;
   END_VAR
BEGIN


   REGION "FOR EACH STATION"
       FOR #i := 0 TO "stnCount" DO

           REGION "FOR EACH BUTTON"
               FOR #j := 1 TO "ptsPerStn" DO

                   REGION "COPY TO LOCAL"
                       #partReq := #stations.me[#i].btnStates[#j];
                       #oldPartReq := #old.partReq.me[#i, #j];
                   END_REGION

                   REGION "DETERMINE STATE"

                       REGION "PART REQUEST FALLING EDGE"
                           IF NOT #partReq AND #oldPartReq THEN

                               REGION "COPY TO LOCAL"
                                   #partNumber := #stations.me[#i].partNumbers[#j];
                               END_REGION

                               REGION "BUTTON HAS NO PART"
                                   IF #partNumber = wstring#'' THEN
                                       #hasPart := FALSE;
                                       #noPart := TRUE;
                                   END_IF;
                               END_REGION

                               REGION "BUTTON HAS PART"
                                   IF #partNumber <> wstring#'' THEN
                                       #hasPart := TRUE;
                                       #noPart := FALSE;
                                   END_IF;
                               END_REGION

                           END_IF;

                           REGION "SAVE FOR CHANGE DETECTION"
                               #old.partReq.me[#i, #j] := #partReq;
                           END_REGION

                       END_REGION

                   END_REGION

                   REGION "NO PART"
                       IF #noPart THEN

                           REGION "TURN OFF THE LIGHTS"
                               #hasPart := FALSE;
                               #noPart := FALSE;
                           END_REGION

                       END_IF;

                   END_REGION

                   REGION "HAS PART"
                       IF #hasPart THEN

                           REGION "TURN OFF THE LIGHTS"
                               #hasPart := FALSE;
                           END_REGION

                           REGION "CALCULATE ADDRESS"
                               #address := (INT_TO_UINT(#i) + 1) * 10 + (INT_TO_UINT(#j) + 1);
                           END_REGION

                           REGION "RESET FLAG"
                               #removeAddress := FALSE;
                           END_REGION

                           REGION "SEARCH EACH ROW IN PART DB"
                               FOR #k := 0 TO "partReqDataRowCount" DO

                                   REGION "COPY TO LOCAL"
                                       #logAddress := #requests.row[#k].address;
                                   END_REGION

                                   REGION "ON MATCH"
                                       IF #logAddress = #address THEN

                                           REGION "SET FLAG"
                                               #removeAddress := TRUE;
                                           END_REGION

                                           REGION "SAVE POINTER"
                                               #pRemoveRow := #k;
                                           END_REGION

                                       END_IF;
                                   END_REGION

                               END_FOR;
                           END_REGION

                       END_IF;
                   END_REGION

                   REGION "REMOVE ADDRESS"
                       IF #removeAddress THEN

                           REGION "TURN OFF THE LIGHTS"
                               #removeAddress := FALSE;
                           END_REGION

                           REGION "TURN OFF REQUEST"
                               #stations.me[#i].partRequested[#j] := FALSE;
                           END_REGION

                           REGION "REMOVAL PROCESS"

                               REGION "REMOVE ROW"
                                   #requests.row[#pRemoveRow] := #blankRow;
                                   #reqCollapse := TRUE;
                               END_REGION

                               REGION "REMOVE PART ORDERED"
                                   #stations.me[#i].partOrdered[#j] := FALSE;
                               END_REGION

                           END_REGION

                           REGION "ROW POINTER"

                               REGION "DECREMENT"
                                   #pRow := #pRow - 1;
                               END_REGION

                               REGION "LOW LIMIT ROLL OVER"
                                   IF #pRow < 0 THEN
                                       #pRow := 0;
                                   END_IF;
                               END_REGION

                           END_REGION

                       END_IF;
                   END_REGION

               END_FOR;

           END_REGION

       END_FOR;
   END_REGION
END_FUNCTION_BLOCK

FUNCTION_BLOCK "HMI Settings Screen"   // FB14, LAD
{ S7_Optimized_Access := 'TRUE' }
VERSION : 0.1
   VAR_IN_OUT
      settings : "Settings";
      stations : "Stations";
   END_VAR
   VAR
      tmrTimeOut : TON_TIME;
      instStaSel : "Station Selection";
      instKP8BtnSel : "KP8 Button Selections";
      old : Struct
         asgnPN : Bool;
         asgnAlloted : Bool;
         asgnCritical : Bool;
         nextPress : Bool;
         prevPress : Bool;
         selBtnCount : Int;
         selBtnNumber : Int;
         selStnCount : Int;
         selStnNumber : Int;
      END_STRUCT;
      instAsnBtnPrms : "Assign Button Parameters";
      instAniPNTmr : "Animate: PN & Timers";
   END_VAR
   VAR_TEMP
      pBN : Int;
      pSN : Int;
      wStringBox : WString;
   END_VAR
   VAR CONSTANT
      ptTimeOut : Time := t#15m;
   END_VAR
   VAR_TEMP   // added for the SCL form of the ladder/FBD networks
      _w1 : Bool;
   END_VAR
BEGIN

REGION Network 1: ENTRY TIMEOUT
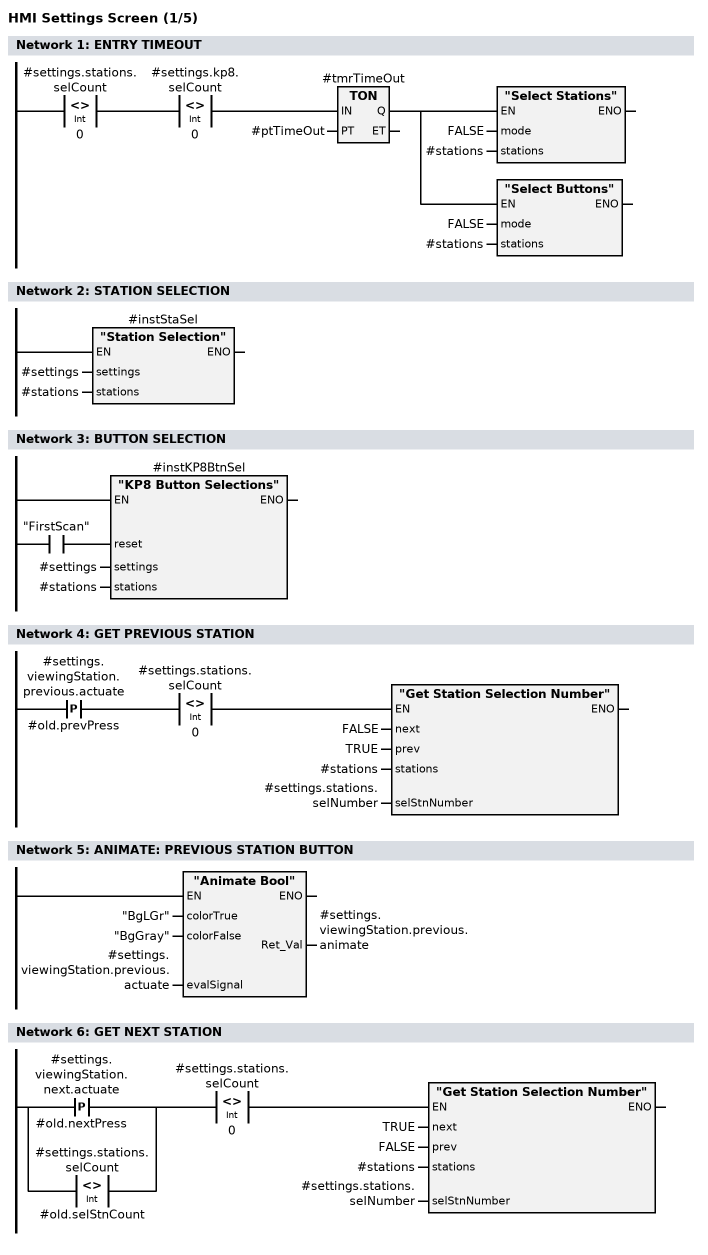
   #tmrTimeOut(IN := (#settings.stations.selCount <> 0) AND (#settings.kp8.selCount <> 0), PT := #ptTimeOut);   // TON
   IF #tmrTimeOut.Q THEN
       "Select Stations"(mode := FALSE, stations := #stations);
       "Select Buttons"(mode := FALSE, stations := #stations);
   END_IF;
END_REGION

REGION Network 2: STATION SELECTION
   RUNG wire#powerrail
      #instStaSel(settings := #settings, stations := #stations)
   END_RUNG
   // the same network as SCL:
   #instStaSel(settings := #settings, stations := #stations);   // "Station Selection"
END_REGION

REGION Network 3: BUTTON SELECTION
   RUNG wire#powerrail
      #instKP8BtnSel(reset := wire#w1, settings := #settings, stations := #stations)
   END_RUNG
   RUNG wire#powerrail
      Contact( "FirstScan" )
   END_RUNG wire#w1
   // the same network as SCL:
   #instKP8BtnSel(reset := "FirstScan", settings := #settings, stations := #stations);   // "KP8 Button Selections"
END_REGION

REGION Network 4: GET PREVIOUS STATION
   RUNG wire#powerrail
      P_Contact(operand := #settings.viewingStation.previous.actuate, bit := #old.prevPress)
      { S7_Templates := "SrcType := Int" } NE_Contact(in1 := #settings.stations.selCount, in2 := 0)
      "Get Station Selection Number"(next := FALSE, prev := TRUE, stations := #stations, selStnNumber := #settings.stations.selNumber)
   END_RUNG
   // the same network as SCL:
   #_w1 := #settings.viewingStation.previous.actuate AND NOT #old.prevPress;   // rising edge of #settings.viewingStation.previous.actuate
   #old.prevPress := #settings.viewingStation.previous.actuate;
   IF #_w1 AND (#settings.stations.selCount <> 0) THEN
       "Get Station Selection Number"(next := FALSE,
                               prev := TRUE,
                               stations := #stations,
                               selStnNumber := #settings.stations.selNumber);
   END_IF;
END_REGION

REGION Network 5: ANIMATE: PREVIOUS STATION BUTTON
   RUNG wire#powerrail
      "Animate Bool"(colorTrue := "BgLGr", colorFalse := "BgGray", evalSignal := #settings.viewingStation.previous.actuate, Ret_Val => #settings.viewingStation.previous.animate)
   END_RUNG
   // the same network as SCL:
   #settings.viewingStation.previous.animate := "Animate Bool"(colorTrue := "BgLGr",
                           colorFalse := "BgGray",
                           evalSignal := #settings.viewingStation.previous.actuate);
END_REGION

REGION Network 6: GET NEXT STATION
   RUNG wire#powerrail
      P_Contact(operand := #settings.viewingStation.next.actuate, bit := #old.nextPress)
      wire#w1
      { S7_Templates := "SrcType := Int" } NE_Contact(in1 := #settings.stations.selCount, in2 := 0)
      "Get Station Selection Number"(next := TRUE, prev := FALSE, stations := #stations, selStnNumber := #settings.stations.selNumber)
   END_RUNG
   RUNG wire#powerrail
      { S7_Templates := "SrcType := Int" } NE_Contact(in1 := #settings.stations.selCount, in2 := #old.selStnCount)
   END_RUNG wire#w1
   // the same network as SCL:
   #_w1 := #settings.viewingStation.next.actuate AND NOT #old.nextPress;   // rising edge of #settings.viewingStation.next.actuate
   #old.nextPress := #settings.viewingStation.next.actuate;
   IF (#_w1 OR (#settings.stations.selCount <> #old.selStnCount)) AND (#settings.stations.selCount <> 0) THEN
       "Get Station Selection Number"(next := TRUE,
                               prev := FALSE,
                               stations := #stations,
                               selStnNumber := #settings.stations.selNumber);
   END_IF;
END_REGION

REGION Network 7: ANIMATE: NEXT STATION BUTTON
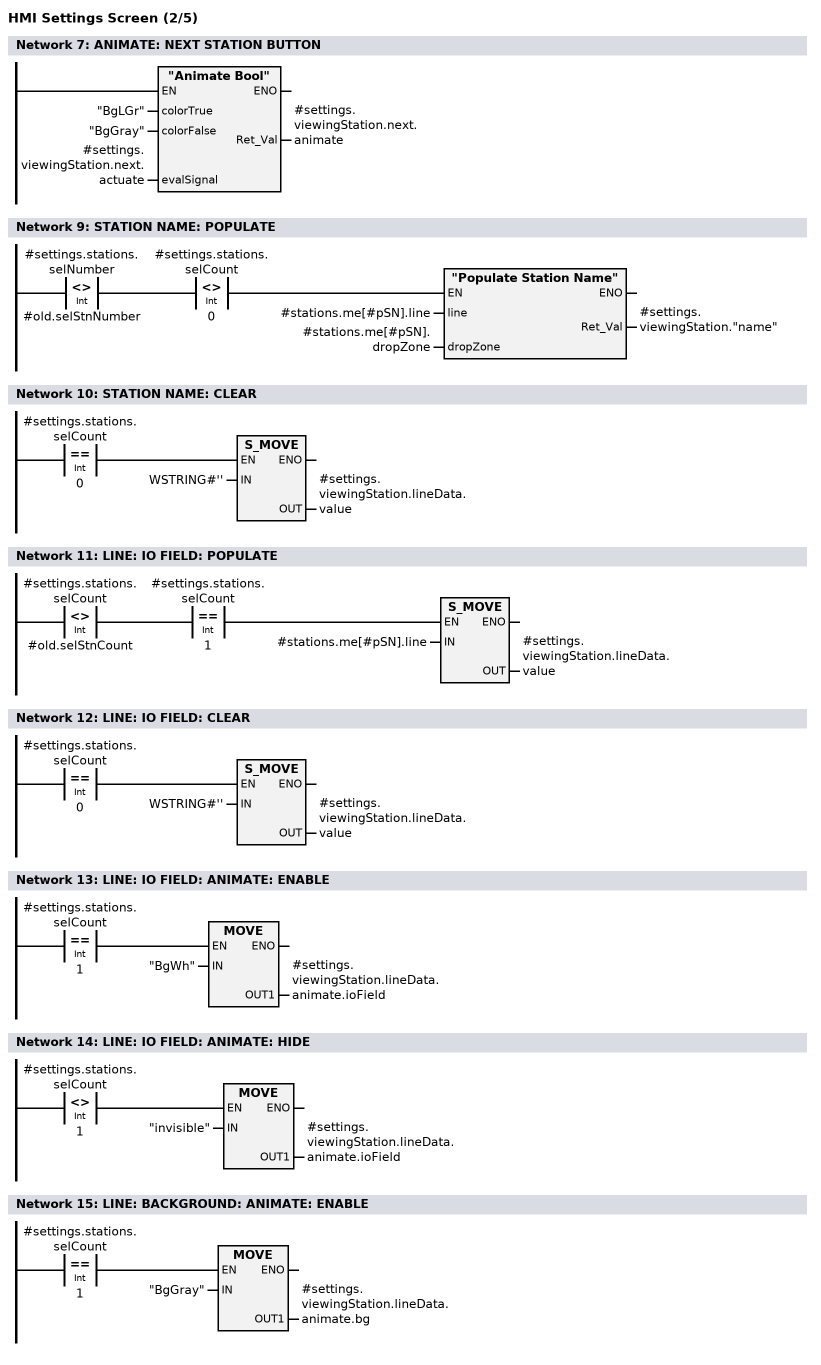
   RUNG wire#powerrail
      "Animate Bool"(colorTrue := "BgLGr", colorFalse := "BgGray", evalSignal := #settings.viewingStation.next.actuate, Ret_Val => #settings.viewingStation.next.animate)
   END_RUNG
   // the same network as SCL:
   #settings.viewingStation.next.animate := "Animate Bool"(colorTrue := "BgLGr",
                           colorFalse := "BgGray",
                           evalSignal := #settings.viewingStation.next.actuate);
END_REGION

REGION Network 8 (SCL): COPY TO POINTERS
   #pSN := #settings.stations.selNumber;
   #pBN := #settings.kp8.selBtnNumber;
END_REGION

REGION Network 9: STATION NAME: POPULATE
   RUNG wire#powerrail
      { S7_Templates := "SrcType := Int" } NE_Contact(in1 := #settings.stations.selNumber, in2 := #old.selStnNumber)
      { S7_Templates := "SrcType := Int" } NE_Contact(in1 := #settings.stations.selCount, in2 := 0)
      "Populate Station Name"(line := #stations.me[#pSN].line, dropZone := #stations.me[#pSN].dropZone, Ret_Val => #settings.viewingStation."name")
   END_RUNG
   // the same network as SCL:
   IF (#settings.stations.selNumber <> #old.selStnNumber) AND (#settings.stations.selCount <> 0) THEN
       #settings.viewingStation."name" := "Populate Station Name"(line := #stations.me[#pSN].line,
                               dropZone := #stations.me[#pSN].dropZone);
   END_IF;
END_REGION

REGION Network 10: STATION NAME: CLEAR
   RUNG wire#powerrail
      { S7_Templates := "SrcType := Int" } EQ_Contact(in1 := #settings.stations.selCount, in2 := 0)
      S_Move(in := WSTRING#'', out => #settings.viewingStation.lineData.value)
   END_RUNG
   // the same network as SCL:
   IF #settings.stations.selCount = 0 THEN #settings.viewingStation.lineData.value := WSTRING#''; END_IF;
END_REGION

REGION Network 11: LINE: IO FIELD: POPULATE
   RUNG wire#powerrail
      { S7_Templates := "SrcType := Int" } NE_Contact(in1 := #settings.stations.selCount, in2 := #old.selStnCount)
      { S7_Templates := "SrcType := Int" } EQ_Contact(in1 := #settings.stations.selCount, in2 := 1)
      S_Move(in := #stations.me[#pSN].line, out => #settings.viewingStation.lineData.value)
   END_RUNG
   // the same network as SCL:
   IF (#settings.stations.selCount <> #old.selStnCount) AND (#settings.stations.selCount = 1) THEN
       #settings.viewingStation.lineData.value := #stations.me[#pSN].line;
   END_IF;
END_REGION

REGION Network 12: LINE: IO FIELD: CLEAR
   RUNG wire#powerrail
      { S7_Templates := "SrcType := Int" } EQ_Contact(in1 := #settings.stations.selCount, in2 := 0)
      S_Move(in := WSTRING#'', out => #settings.viewingStation.lineData.value)
   END_RUNG
   // the same network as SCL:
   IF #settings.stations.selCount = 0 THEN #settings.viewingStation.lineData.value := WSTRING#''; END_IF;
END_REGION

REGION Network 13: LINE: IO FIELD: ANIMATE: ENABLE
   RUNG wire#powerrail
      { S7_Templates := "SrcType := Int" } EQ_Contact(in1 := #settings.stations.selCount, in2 := 1)
      Move(in := "BgWh", out1 => #settings.viewingStation.lineData.animate.ioField)
   END_RUNG
   // the same network as SCL:
   IF #settings.stations.selCount = 1 THEN
       #settings.viewingStation.lineData.animate.ioField := "BgWh";
   END_IF;
END_REGION

REGION Network 14: LINE: IO FIELD: ANIMATE: HIDE
   RUNG wire#powerrail
      { S7_Templates := "SrcType := Int" } NE_Contact(in1 := #settings.stations.selCount, in2 := 1)
      Move(in := "invisible", out1 => #settings.viewingStation.lineData.animate.ioField)
   END_RUNG
   // the same network as SCL:
   IF #settings.stations.selCount <> 1 THEN
       #settings.viewingStation.lineData.animate.ioField := "invisible";
   END_IF;
END_REGION

REGION Network 15: LINE: BACKGROUND: ANIMATE: ENABLE
   RUNG wire#powerrail
      { S7_Templates := "SrcType := Int" } EQ_Contact(in1 := #settings.stations.selCount, in2 := 1)
      Move(in := "BgGray", out1 => #settings.viewingStation.lineData.animate.bg)
   END_RUNG
   // the same network as SCL:
   IF #settings.stations.selCount = 1 THEN #settings.viewingStation.lineData.animate.bg := "BgGray"; END_IF;
END_REGION

REGION Network 16: LINE: BACKGROUND: ANIMATE: HIDE
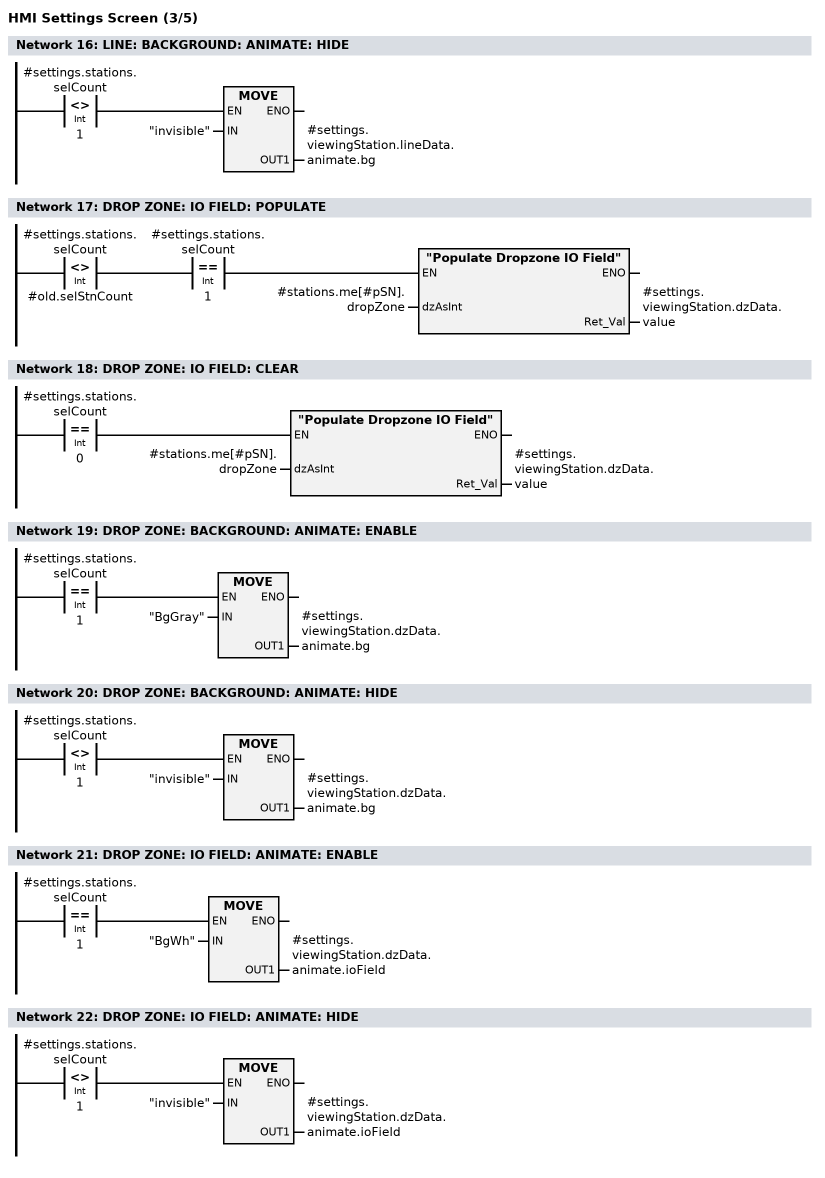
   RUNG wire#powerrail
      { S7_Templates := "SrcType := Int" } NE_Contact(in1 := #settings.stations.selCount, in2 := 1)
      Move(in := "invisible", out1 => #settings.viewingStation.lineData.animate.bg)
   END_RUNG
   // the same network as SCL:
   IF #settings.stations.selCount <> 1 THEN
       #settings.viewingStation.lineData.animate.bg := "invisible";
   END_IF;
END_REGION

REGION Network 17: DROP ZONE: IO FIELD: POPULATE
   RUNG wire#powerrail
      { S7_Templates := "SrcType := Int" } NE_Contact(in1 := #settings.stations.selCount, in2 := #old.selStnCount)
      { S7_Templates := "SrcType := Int" } EQ_Contact(in1 := #settings.stations.selCount, in2 := 1)
      "Populate Dropzone IO Field"(dzAsInt := #stations.me[#pSN].dropZone, Ret_Val => #settings.viewingStation.dzData.value)
   END_RUNG
   // the same network as SCL:
   IF (#settings.stations.selCount <> #old.selStnCount) AND (#settings.stations.selCount = 1) THEN
       #settings.viewingStation.dzData.value := "Populate Dropzone IO Field"(dzAsInt := #stations.me[#pSN].dropZone);
   END_IF;
END_REGION

REGION Network 18: DROP ZONE: IO FIELD: CLEAR
   RUNG wire#powerrail
      { S7_Templates := "SrcType := Int" } EQ_Contact(in1 := #settings.stations.selCount, in2 := 0)
      "Populate Dropzone IO Field"(dzAsInt := #stations.me[#pSN].dropZone, Ret_Val => #settings.viewingStation.dzData.value)
   END_RUNG
   // the same network as SCL:
   IF #settings.stations.selCount = 0 THEN
       #settings.viewingStation.dzData.value := "Populate Dropzone IO Field"(dzAsInt := #stations.me[#pSN].dropZone);
   END_IF;
END_REGION

REGION Network 19: DROP ZONE: BACKGROUND: ANIMATE: ENABLE
   RUNG wire#powerrail
      { S7_Templates := "SrcType := Int" } EQ_Contact(in1 := #settings.stations.selCount, in2 := 1)
      Move(in := "BgGray", out1 => #settings.viewingStation.dzData.animate.bg)
   END_RUNG
   // the same network as SCL:
   IF #settings.stations.selCount = 1 THEN #settings.viewingStation.dzData.animate.bg := "BgGray"; END_IF;
END_REGION

REGION Network 20: DROP ZONE: BACKGROUND: ANIMATE: HIDE
   RUNG wire#powerrail
      { S7_Templates := "SrcType := Int" } NE_Contact(in1 := #settings.stations.selCount, in2 := 1)
      Move(in := "invisible", out1 => #settings.viewingStation.dzData.animate.bg)
   END_RUNG
   // the same network as SCL:
   IF #settings.stations.selCount <> 1 THEN
       #settings.viewingStation.dzData.animate.bg := "invisible";
   END_IF;
END_REGION

REGION Network 21: DROP ZONE: IO FIELD: ANIMATE: ENABLE
   RUNG wire#powerrail
      { S7_Templates := "SrcType := Int" } EQ_Contact(in1 := #settings.stations.selCount, in2 := 1)
      Move(in := "BgWh", out1 => #settings.viewingStation.dzData.animate.ioField)
   END_RUNG
   // the same network as SCL:
   IF #settings.stations.selCount = 1 THEN #settings.viewingStation.dzData.animate.ioField := "BgWh"; END_IF;
END_REGION

REGION Network 22: DROP ZONE: IO FIELD: ANIMATE: HIDE
   RUNG wire#powerrail
      { S7_Templates := "SrcType := Int" } NE_Contact(in1 := #settings.stations.selCount, in2 := 1)
      Move(in := "invisible", out1 => #settings.viewingStation.dzData.animate.ioField)
   END_RUNG
   // the same network as SCL:
   IF #settings.stations.selCount <> 1 THEN
       #settings.viewingStation.dzData.animate.ioField := "invisible";
   END_IF;
END_REGION

REGION Network 23: PART NUMBER IO FIELD: POPULATE
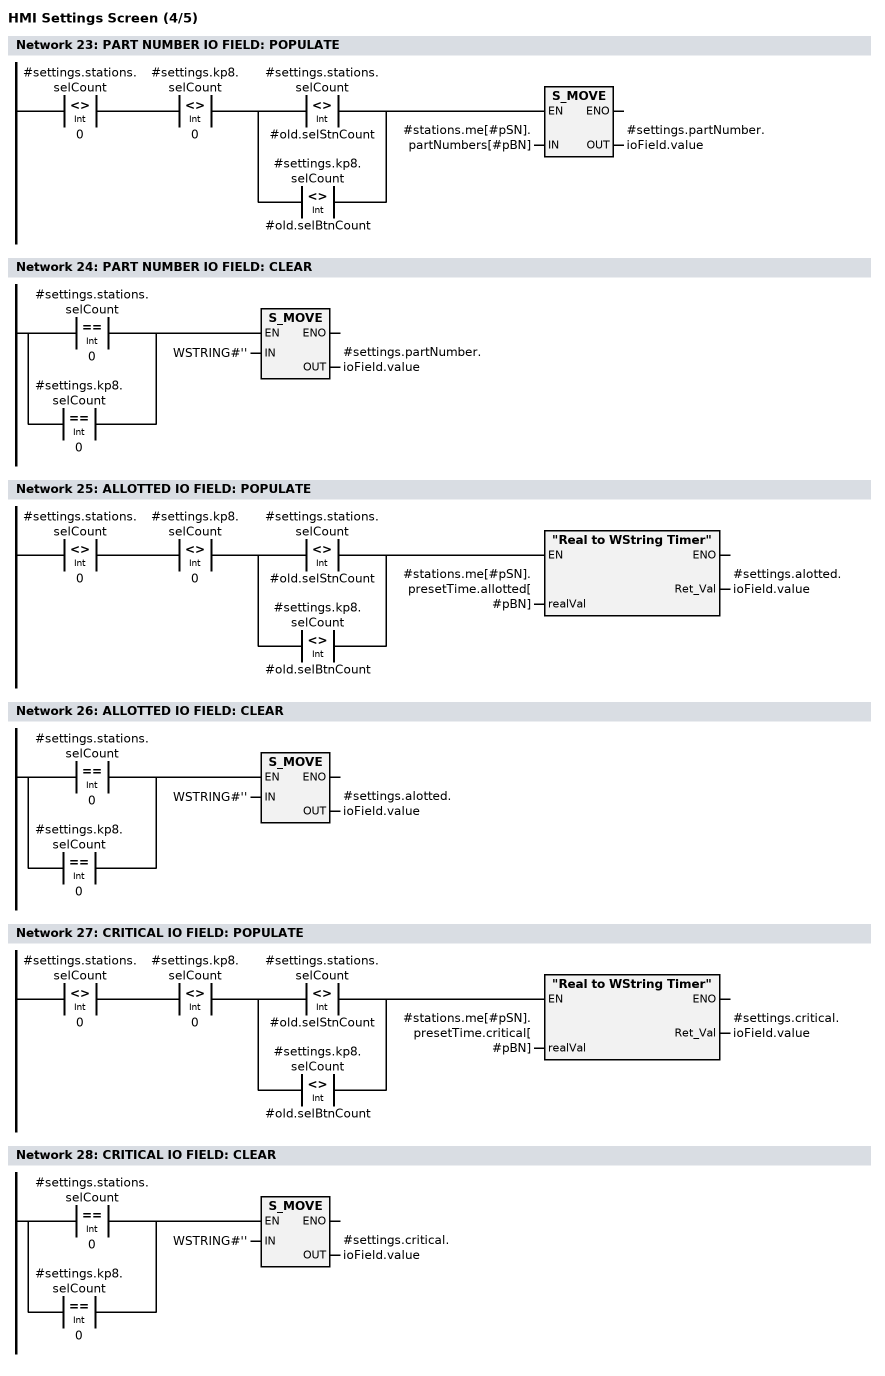
   RUNG wire#powerrail
      { S7_Templates := "SrcType := Int" } NE_Contact(in1 := #settings.stations.selCount, in2 := 0)
      { S7_Templates := "SrcType := Int" } NE_Contact(in1 := #settings.kp8.selCount, in2 := 0)
      wire#w1
      { S7_Templates := "SrcType := Int" } NE_Contact(in1 := #settings.stations.selCount, in2 := #old.selStnCount)
      wire#w2
      S_Move(in := #stations.me[#pSN].partNumbers[#pBN], out => #settings.partNumber.ioField.value)
   END_RUNG
   RUNG wire#w1
      { S7_Templates := "SrcType := Int" } NE_Contact(in1 := #settings.kp8.selCount, in2 := #old.selBtnCount)
   END_RUNG wire#w2
   // the same network as SCL:
   IF (#settings.stations.selCount <> 0) AND (#settings.kp8.selCount <> 0) AND ((#settings.stations.selCount <> #old.selStnCount) OR (#settings.kp8.selCount <> #old.selBtnCount)) THEN
       #settings.partNumber.ioField.value := #stations.me[#pSN].partNumbers[#pBN];
   END_IF;
END_REGION

REGION Network 24: PART NUMBER IO FIELD: CLEAR
   RUNG wire#powerrail
      { S7_Templates := "SrcType := Int" } EQ_Contact(in1 := #settings.stations.selCount, in2 := 0)
      wire#w1
      S_Move(in := WSTRING#'', out => #settings.partNumber.ioField.value)
   END_RUNG
   RUNG wire#powerrail
      { S7_Templates := "SrcType := Int" } EQ_Contact(in1 := #settings.kp8.selCount, in2 := 0)
   END_RUNG wire#w1
   // the same network as SCL:
   IF (#settings.stations.selCount = 0) OR (#settings.kp8.selCount = 0) THEN
       #settings.partNumber.ioField.value := WSTRING#'';
   END_IF;
END_REGION

REGION Network 25: ALLOTTED IO FIELD: POPULATE
   RUNG wire#powerrail
      { S7_Templates := "SrcType := Int" } NE_Contact(in1 := #settings.stations.selCount, in2 := 0)
      { S7_Templates := "SrcType := Int" } NE_Contact(in1 := #settings.kp8.selCount, in2 := 0)
      wire#w1
      { S7_Templates := "SrcType := Int" } NE_Contact(in1 := #settings.stations.selCount, in2 := #old.selStnCount)
      wire#w2
      "Real to WString Timer"(realVal := #stations.me[#pSN].presetTime.allotted[#pBN], Ret_Val => #settings.alotted.ioField.value)
   END_RUNG
   RUNG wire#w1
      { S7_Templates := "SrcType := Int" } NE_Contact(in1 := #settings.kp8.selCount, in2 := #old.selBtnCount)
   END_RUNG wire#w2
   // the same network as SCL:
   IF (#settings.stations.selCount <> 0) AND (#settings.kp8.selCount <> 0) AND ((#settings.stations.selCount <> #old.selStnCount) OR (#settings.kp8.selCount <> #old.selBtnCount)) THEN
       #settings.alotted.ioField.value := "Real to WString Timer"(realVal := #stations.me[#pSN].presetTime.allotted[#pBN]);
   END_IF;
END_REGION

REGION Network 26: ALLOTTED IO FIELD: CLEAR
   RUNG wire#powerrail
      { S7_Templates := "SrcType := Int" } EQ_Contact(in1 := #settings.stations.selCount, in2 := 0)
      wire#w1
      S_Move(in := WSTRING#'', out => #settings.alotted.ioField.value)
   END_RUNG
   RUNG wire#powerrail
      { S7_Templates := "SrcType := Int" } EQ_Contact(in1 := #settings.kp8.selCount, in2 := 0)
   END_RUNG wire#w1
   // the same network as SCL:
   IF (#settings.stations.selCount = 0) OR (#settings.kp8.selCount = 0) THEN
       #settings.alotted.ioField.value := WSTRING#'';
   END_IF;
END_REGION

REGION Network 27: CRITICAL IO FIELD: POPULATE
   RUNG wire#powerrail
      { S7_Templates := "SrcType := Int" } NE_Contact(in1 := #settings.stations.selCount, in2 := 0)
      { S7_Templates := "SrcType := Int" } NE_Contact(in1 := #settings.kp8.selCount, in2 := 0)
      wire#w1
      { S7_Templates := "SrcType := Int" } NE_Contact(in1 := #settings.stations.selCount, in2 := #old.selStnCount)
      wire#w2
      "Real to WString Timer"(realVal := #stations.me[#pSN].presetTime.critical[#pBN], Ret_Val => #settings.critical.ioField.value)
   END_RUNG
   RUNG wire#w1
      { S7_Templates := "SrcType := Int" } NE_Contact(in1 := #settings.kp8.selCount, in2 := #old.selBtnCount)
   END_RUNG wire#w2
   // the same network as SCL:
   IF (#settings.stations.selCount <> 0) AND (#settings.kp8.selCount <> 0) AND ((#settings.stations.selCount <> #old.selStnCount) OR (#settings.kp8.selCount <> #old.selBtnCount)) THEN
       #settings.critical.ioField.value := "Real to WString Timer"(realVal := #stations.me[#pSN].presetTime.critical[#pBN]);
   END_IF;
END_REGION

REGION Network 28: CRITICAL IO FIELD: CLEAR
   RUNG wire#powerrail
      { S7_Templates := "SrcType := Int" } EQ_Contact(in1 := #settings.stations.selCount, in2 := 0)
      wire#w1
      S_Move(in := WSTRING#'', out => #settings.critical.ioField.value)
   END_RUNG
   RUNG wire#powerrail
      { S7_Templates := "SrcType := Int" } EQ_Contact(in1 := #settings.kp8.selCount, in2 := 0)
   END_RUNG wire#w1
   // the same network as SCL:
   IF (#settings.stations.selCount = 0) OR (#settings.kp8.selCount = 0) THEN
       #settings.critical.ioField.value := WSTRING#'';
   END_IF;
END_REGION

REGION Network 29: PART NUMBER, ALLOTTED & CRITICAL: ANIMATE
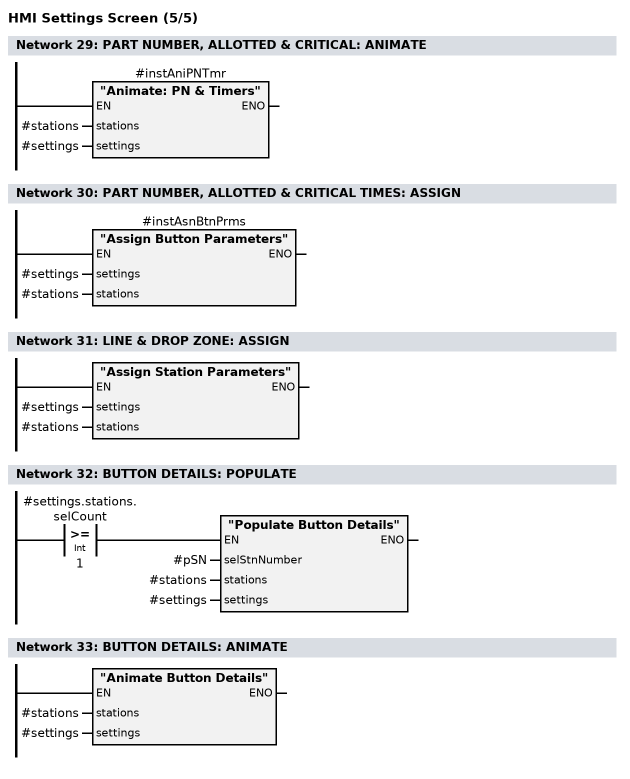
   RUNG wire#powerrail
      #instAniPNTmr(stations := #stations, settings := #settings)
   END_RUNG
   // the same network as SCL:
   #instAniPNTmr(stations := #stations, settings := #settings);   // "Animate: PN & Timers"
END_REGION

REGION Network 30: PART NUMBER, ALLOTTED & CRITICAL TIMES: ASSIGN
   RUNG wire#powerrail
      #instAsnBtnPrms(settings := #settings, stations := #stations)
   END_RUNG
   // the same network as SCL:
   #instAsnBtnPrms(settings := #settings, stations := #stations);   // "Assign Button Parameters"
END_REGION

REGION Network 31: LINE & DROP ZONE: ASSIGN
   RUNG wire#powerrail
      "Assign Station Parameters"(settings := #settings, stations := #stations)
   END_RUNG
   // the same network as SCL:
   "Assign Station Parameters"(settings := #settings, stations := #stations);
END_REGION

REGION Network 32: BUTTON DETAILS: POPULATE
   RUNG wire#powerrail
      { S7_Templates := "SrcType := Int" } GE_Contact(in1 := #settings.stations.selCount, in2 := 1)
      "Populate Button Details"(selStnNumber := #pSN, stations := #stations, settings := #settings)
   END_RUNG
   // the same network as SCL:
   IF #settings.stations.selCount >= 1 THEN
       "Populate Button Details"(selStnNumber := #pSN, stations := #stations, settings := #settings);
   END_IF;
END_REGION

REGION Network 33: BUTTON DETAILS: ANIMATE
   RUNG wire#powerrail
      "Animate Button Details"(stations := #stations, settings := #settings)
   END_RUNG
   // the same network as SCL:
   "Animate Button Details"(stations := #stations, settings := #settings);
END_REGION

REGION Network 34 (SCL): CHANGE DETECTION
   #old.selBtnCount := #settings.kp8.selCount;
   #old.selBtnNumber := #settings.kp8.selBtnNumber;
   #old.selStnCount := #settings.stations.selCount;
   #old.selStnNumber := #settings.stations.selNumber;
END_REGION
END_FUNCTION_BLOCK

FUNCTION_BLOCK "Collapse Table"   // FB15, SCL
{ S7_Optimized_Access := 'TRUE' }
VERSION : 0.1
   VAR_INPUT
      firstScan : Bool;
   END_VAR
   VAR_IN_OUT
      reqCollapse : Bool;
      requests : "Part Request Data";
   END_VAR
   VAR
      tableBox : "Part Request Data";
   END_VAR
   VAR_TEMP
      address : Int;
      blankRow : "Table Row";
      collapseReq : Bool;
      i : Int;
      pCollapse : Int;
      clearItrnlTable : Bool;
   END_VAR
BEGIN
   REGION "CLEAR TABLE REQUESTS"
       IF #firstScan OR #reqCollapse THEN
           #clearItrnlTable := TRUE;
           #reqCollapse := FALSE;
       END_IF;
   END_REGION

   REGION "REMOVE EMPTY ROWS"

       REGION "FOR EACH ROW IN PART DB"
           FOR #i := 0 TO "partReqDataRowCount" DO

               REGION "COPY TO LOCAL"
                   #address := UINT_TO_INT(#requests.row[#i].address);
               END_REGION

               REGION "ROW IS NOT EMPTY"
                   IF #address <> 0 THEN

                       REGION "MOVE TO TEMP TABLE"
                           #tableBox.row[#pCollapse] := #requests.row[#i];
                       END_REGION

                       REGION "CALCULATE POINTER"
                           #pCollapse += 1;
                       END_REGION

                   END_IF;
               END_REGION

               REGION "ROW IS EMPTY"
                   IF #address = 0 THEN

                       REGION "SET FLAG"
                           #collapseReq := TRUE;
                       END_REGION

                   END_IF;
               END_REGION

           END_FOR;
       END_REGION

   END_REGION

   REGION "COLLAPSE TABLE"
       IF #collapseReq THEN

           REGION "TURN OFF THE LIGHTS"
               #collapseReq := FALSE;
           END_REGION

           REGION "COPY TEMP TO PERMANENT"
               #requests := #tableBox;
           END_REGION

           REGION "CLEAR VALUES FROM TEMP TABLE"
               #clearItrnlTable := TRUE;
           END_REGION

       END_IF;
   END_REGION


   REGION "CLEAR VALUES FROM TEMP TABLE"
       IF #clearItrnlTable THEN
           FOR #i := 0 TO "partReqDataRowCount" DO
               #tableBox.row[#i] := #blankRow;
           END_FOR;
       END_IF;
   END_REGION
END_FUNCTION_BLOCK

FUNCTION_BLOCK "HMI Populate Part Call"   // FB16, SCL
{ S7_Optimized_Access := 'TRUE' }
VERSION : 0.1
   VAR_INPUT
      firstScan : Bool;
      currentRowCount : Int;
      requests : "Part Request Data";
   END_VAR
   VAR_IN_OUT
      partCall : "Part Call Screen";
      tableNav : "Table Nav";
   END_VAR
   VAR
      firstRow : Int;
      old : Struct
         top : Bool;
         pgUp : Bool;
         lnUp : Bool;
         lnDn : Bool;
         pgDn : Bool;
         btm : Bool;
      END_STRUCT;
   END_VAR
   VAR_TEMP
      animate : Bool;
      btn : Struct
         top : Bool;
         pgUp : Bool;
         lnUp : Bool;
         lnDn : Bool;
         pgDn : Bool;
         btm : Bool;
      END_STRUCT;
      gray : USInt;
      green : USInt;
      i : Int;
      maxDBRows : Int;
      pRow : Int;
      visibleRows : Int;
      thisRow : Int;
      saveAct : Bool;
   END_VAR
BEGIN
   REGION "COPY TO LOCAL"
       #visibleRows := "partReqHmiRowCount";
       #maxDBRows := #currentRowCount;
       #btn.top := #tableNav.top.actuate;
       #btn.pgUp := #tableNav.pageUp.actuate;
       #btn.lnUp := #tableNav.lineUp.actuate;
       #btn.lnDn := #tableNav.lineDown.actuate;
       #btn.pgDn := #tableNav.pageDown.actuate;
       #btn.btm := #tableNav.bottom.actuate;
   END_REGION

   REGION "RESOLVE FIRST ROW"

       REGION "TOP"
           IF NOT #btn.top AND #old.top THEN
               #firstRow := 0;
           END_IF;
       END_REGION

       REGION "PAGE UP"
           IF NOT #btn.pgUp AND #old.pgUp THEN
               #firstRow -= #visibleRows - 1;
           END_IF;
       END_REGION

       REGION "LINE UP"
           IF NOT #btn.lnUp AND #old.lnUp THEN
               #firstRow -= 1;
           END_IF;
       END_REGION

       REGION "LINE DOWN"
           IF NOT #btn.lnDn AND #old.lnDn THEN
               #firstRow += 1;
           END_IF;
       END_REGION

       REGION "PAGE DOWN"
           IF NOT #btn.pgDn AND #old.pgDn THEN
               #firstRow += #visibleRows - 1;
           END_IF;
       END_REGION

       REGION "BOTTOM"
           IF NOT #btn.btm AND #old.btm THEN
               #firstRow := #maxDBRows - #visibleRows + 1;
           END_IF;
       END_REGION

   END_REGION

   REGION "CHANGE DETECTION"
       #old.top := #btn.top;
       #old.pgUp := #btn.pgUp;
       #old.lnUp := #btn.lnUp;
       #old.lnDn := #btn.lnDn;
       #old.pgDn := #btn.pgDn;
       #old.btm := #btn.btm;
   END_REGION

   REGION "ANIMATE PART CALL NAV"

       REGION "COPY TO LOCAL"
           #gray := "BgGray";
           #green := "BgLGr";
       END_REGION

       REGION "TOP"
           #tableNav.top.animate := "Animate Bool"(colorTrue := #green,
                                                   colorFalse := #gray,
                                                   evalSignal := #tableNav.top.actuate);
       END_REGION

       REGION "PAGE UP"
           #tableNav.pageUp.animate := "Animate Bool"(colorTrue := #green,
                                                      colorFalse := #gray,
                                                      evalSignal := #tableNav.pageUp.actuate);
       END_REGION

       REGION "LINE UP"
           #tableNav.lineUp.animate := "Animate Bool"(colorTrue := #green,
                                                      colorFalse := #gray,
                                                      evalSignal := #tableNav.lineUp.actuate);
       END_REGION

       REGION "LINE DOWN"
           #tableNav.lineDown.animate := "Animate Bool"(colorTrue := #green,
                                                        colorFalse := #gray,
                                                        evalSignal := #tableNav.lineDown.actuate);
       END_REGION

       REGION "PAGE DOWN"
           #tableNav.pageDown.animate := "Animate Bool"(colorTrue := #green,
                                                        colorFalse := #gray,
                                                        evalSignal := #tableNav.pageDown.actuate);
       END_REGION

       REGION "BOTTOM"
           #tableNav.bottom.animate := "Animate Bool"(colorTrue := #green,
                                                      colorFalse := #gray,
                                                      evalSignal := #tableNav.bottom.actuate);
       END_REGION

   END_REGION

   REGION "UPPER LIMIT ROLL OVER"
       IF #firstRow > #maxDBRows THEN
           #firstRow -= #maxDBRows - 1;
       END_IF;
   END_REGION

   REGION "LOWER LIMIT ROLL OVER"
       IF #firstRow < 0 THEN
           #firstRow += #maxDBRows - 1;
       END_IF;
   END_REGION

   REGION "LOOP THROUGH DISPLAYED STATIONS"
       FOR #i := 0 TO #visibleRows - 1 DO

           REGION "CALCULATE POINTER"
               #pRow := #firstRow + #i;
           END_REGION

           REGION "UPPER LIMIT ROLL OVER"
               IF #maxDBRows <= #visibleRows THEN
                   #pRow := #i;
               END_IF;
               IF #pRow >= #maxDBRows AND #maxDBRows >= #visibleRows THEN
                   #pRow := #firstRow + #i - #maxDBRows;
               END_IF;
           END_REGION

           REGION "SEND TO HMI"
               #saveAct := #partCall.row[#i].pbSelection.actuate;
               #partCall.row[#i] := #requests.row[#pRow];
               #partCall.row[#i].pbSelection.actuate := #saveAct;
           END_REGION

       END_FOR;
   END_REGION
END_FUNCTION_BLOCK

FUNCTION_BLOCK "Clear Part Requests"   // FB17, SCL
{ S7_Optimized_Access := 'TRUE' }
VERSION : 0.1
   VAR_INPUT
      clearRequest : Bool;
   END_VAR
   VAR_IN_OUT
      requests : "Part Request Data";
      partCall : "Part Call Screen";
      currentRowCount : Int;
   END_VAR
   VAR_TEMP
      blankRow : "Table Row";
      i : Int;
   END_VAR
BEGIN
   REGION "ON REQUEST"
       IF #clearRequest THEN

           REGION "HMI TABLE"

               REGION "CLEAR ROWS"
                   FOR #i := 0 TO "partReqHmiRowCount" DO
                       #partCall.row[#i] := #blankRow;
                   END_FOR;
               END_REGION

           END_REGION

           REGION "PART REQUEST DATA BASE"

               REGION "CLEAR ROWS"
                   FOR #i := 0 TO "partReqDataRowCount" DO
                       #requests.row[#i] := #blankRow;
                       #currentRowCount := 0;
                   END_FOR;
               END_REGION

           END_REGION

       END_IF;
   END_REGION
END_FUNCTION_BLOCK

FUNCTION_BLOCK "Load Default Timer Presets"   // FB18, SCL
{ S7_Optimized_Access := 'TRUE' }
VERSION : 0.1
   VAR_INPUT
      req : Bool;
   END_VAR
   VAR_IN_OUT
      stations : "Stations";
   END_VAR
   VAR
      oldReq : Bool;
   END_VAR
   VAR_TEMP
      alotted : Real;
      critical : Real;
      i : Int;
      j : Int;
      partNumber : WString;
      tmrReal : Real;
   END_VAR
BEGIN
   REGION "COPY TO LOCAL"
       #alotted := "defaultAlotted";
       #critical := "defaultCritical";
   END_REGION

   REGION "ON REQUEST RISING EDGE"
       IF #req AND NOT #oldReq THEN

           REGION "LOOP THROUGH STATIONS" 
               FOR #i := 0 TO "stnCount" DO

                   REGION "LOOP THROUGH BUTTONS"
                       FOR #j := 0 TO "ptsPerStn" DO

                           REGION "COPY TO LOCAL"
                               #partNumber := #stations.me[#i].partNumbers[#j];
                           END_REGION

                           REGION "IF BUTTON HAS ASSOCIATED PN"
                               IF LEN(#partNumber) <> 0 THEN

                                   REGION "COPY TO LOCAL"
                                       #tmrReal := #stations.me[#i].presetTime.allotted[#j];
                                   END_REGION

                                   REGION "ON NO TIME ENTERED"
                                       IF #tmrReal = 0.0 THEN

                                           REGION "ASSIGN ALLOTTED VALUES"
                                               #stations.me[#i].presetTime.allotted[#j] := #alotted;
                                           END_REGION

                                       END_IF;
                                   END_REGION

                                   REGION "COPY TO LOCAL"
                                       #tmrReal := #stations.me[#i].presetTime.critical[#j];
                                   END_REGION

                                   REGION "ON NO TIME ENTERED"
                                       IF #tmrReal = 0.0 THEN

                                           REGION "ASSIGN CRITICAL VALUES"
                                               #stations.me[#i].presetTime.critical[#j] := #critical;
                                           END_REGION

                                       END_IF;
                                   END_REGION

                               END_IF;
                           END_REGION

                       END_FOR;
                   END_REGION

               END_FOR;
           END_REGION

       END_IF;
   END_REGION

   REGION "CHANGE DETECTION"
       #oldReq := #req;
   END_REGION ;
END_FUNCTION_BLOCK

FUNCTION_BLOCK "LED Populate Sign"   // FB19, SCL
{ S7_Optimized_Access := 'TRUE' }
VERSION : 0.1
   VAR_INPUT
      requests : "Part Request Data";
   END_VAR
   VAR_IN_OUT
      ledData : "LED Sign Data";
   END_VAR
   VAR_TEMP
      animate : USInt;
      i : Int;
      visibleRows : Int;
      tempRow : "Table Row";
   END_VAR
BEGIN
   REGION "COPY TO LOCAL"
       #visibleRows := "ledRowCount";
   END_REGION

   REGION "POPULATE SIGN DATA"

       REGION "FOR EACH ROW ON SIGN"
           FOR #i := 0 TO #visibleRows DO

               REGION "GET ROW"
                   #tempRow := #requests.row[#i];
               END_REGION

               REGION "LINE LABEL DARK MODE"                
                   "Dark Mode"(#tempRow.tfLine.animate);
               END_REGION

               REGION "DROP ZONE DARK MODE"
                   "Dark Mode"(#tempRow.tfDropZone.animate);
               END_REGION

               REGION "PART NUMBER DARK MODE"

                   REGION "SINGLE LINE"
                       "Dark Mode"(#tempRow.tfPartNumber.animateSL);
                   END_REGION

                   REGION "DOUBLE LINE"
                       "Dark Mode"(#tempRow.tfPartNumber.animateDL);
                   END_REGION

               END_REGION

               REGION "TIME DARK MODE"
                   "Dark Mode"(#tempRow.tfTime.animate);
               END_REGION

               REGION "SEND TO SIGN"
                   #ledData.row[#i] := #tempRow;
               END_REGION

           END_FOR;
       END_REGION

   END_REGION
END_FUNCTION_BLOCK

